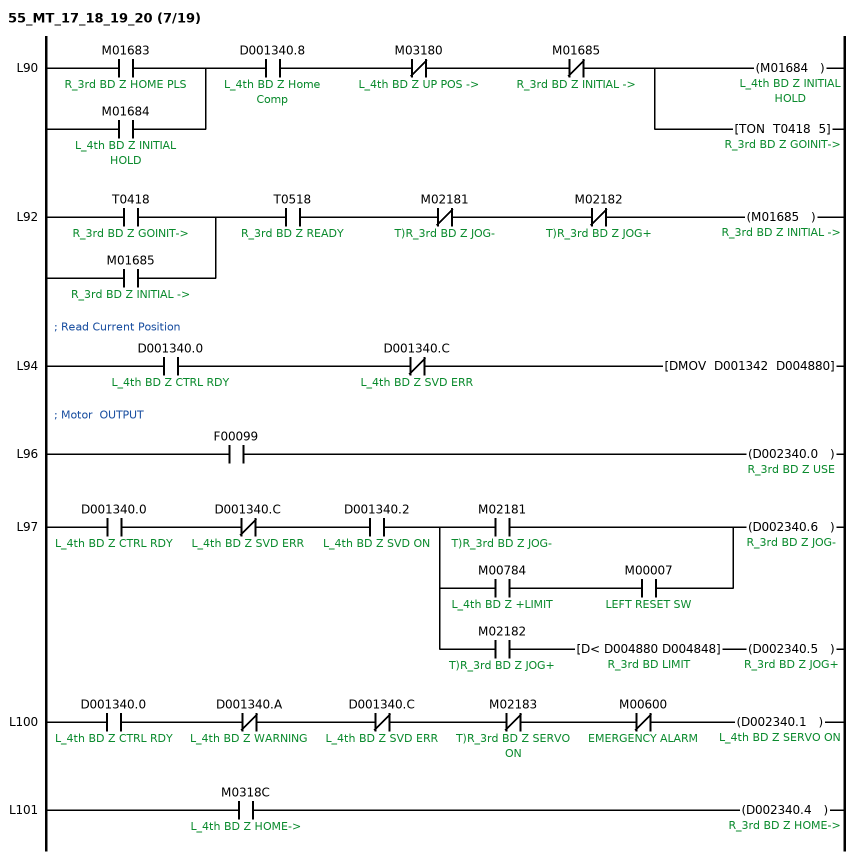
[picture p312: 55_MT_17_18_19_20 rungs L90-L101]
; L90
LOAD      M01683	// R_3rd BD Z HOME PLS
OR        M01684	// L_4th BD Z INITIAL HOLD
AND       D001340.8	// L_4th BD Z Home Comp
AND NOT   M03180	// L_4th BD Z UP POS ->
AND NOT   M01685	// R_3rd BD Z INITIAL ->
OUT       M01684	// L_4th BD Z INITIAL HOLD
TON       T0418 5	// R_3rd BD Z GOINIT->
; L92
LOAD      T0418	// R_3rd BD Z GOINIT->
OR        M01685	// R_3rd BD Z INITIAL ->
AND       T0518	// R_3rd BD Z READY
AND NOT   M02181	// T)R_3rd BD Z JOG-
AND NOT   M02182	// T)R_3rd BD Z JOG+
OUT       M01685	// R_3rd BD Z INITIAL ->
; L94
LOAD      D001340.0	// L_4th BD Z CTRL RDY
AND NOT   D001340.C	// L_4th BD Z SVD ERR
DMOV      D001342 D004880
// output comment: Read Current Position
//  Motor  OUTPUT
; L96
LOAD      F00099
OUT       D002340.0	// R_3rd BD Z USE
; L97
LOAD      D001340.0	// L_4th BD Z CTRL RDY
AND NOT   D001340.C	// L_4th BD Z SVD ERR
AND       D001340.2	// L_4th BD Z SVD ON
MPUSH
LOAD      M02181	// T)R_3rd BD Z JOG-
LOAD      M00784	// L_4th BD Z +LIMIT
AND       M00007	// LEFT RESET SW
OR LOAD
AND LOAD
OUT       D002340.6	// R_3rd BD Z JOG-
MPOP
AND       M02182	// T)R_3rd BD Z JOG+
ANDD<     D004880 D004848	// R_3rd BD LIMIT
OUT       D002340.5	// R_3rd BD Z JOG+
; L100
LOAD      D001340.0	// L_4th BD Z CTRL RDY
AND NOT   D001340.A	// L_4th BD Z WARNING
AND NOT   D001340.C	// L_4th BD Z SVD ERR
AND NOT   M02183	// T)R_3rd BD Z SERVO ON
AND NOT   M00600	// EMERGENCY ALARM
OUT       D002340.1	// L_4th BD Z SERVO ON
; L101
LOAD      M0318C	// L_4th BD Z HOME->
OUT       D002340.4	// R_3rd BD Z HOME->

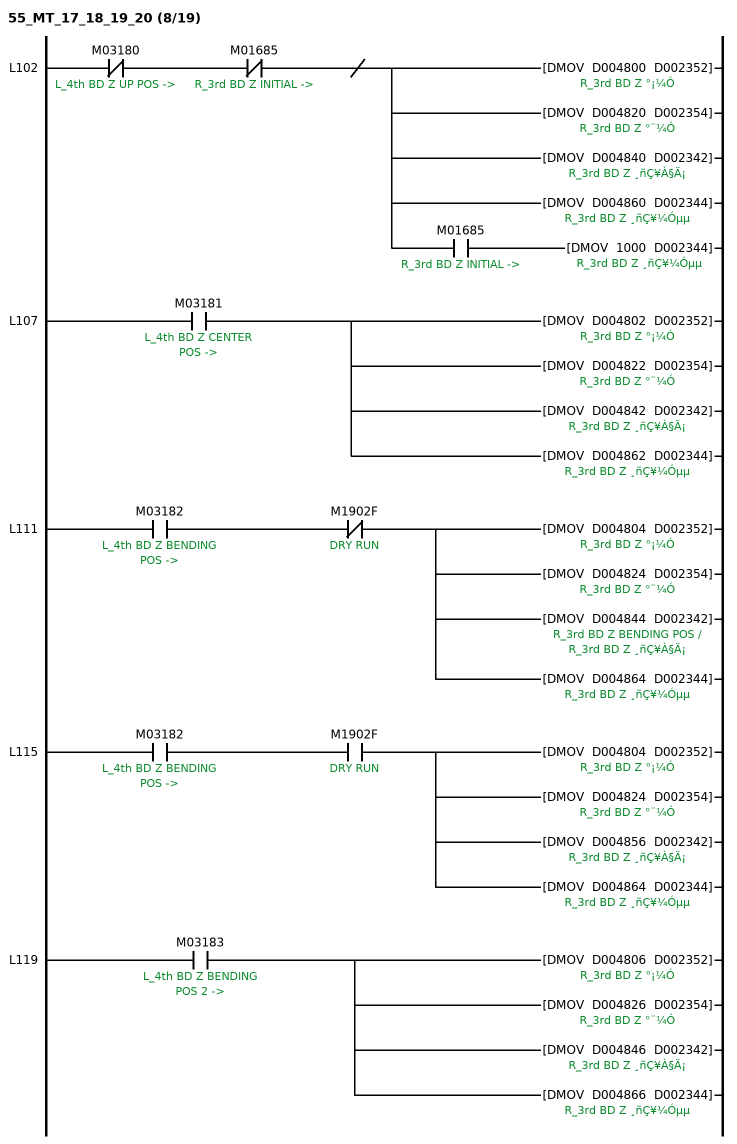
; L102
LOAD NOT  M03180	// L_4th BD Z UP POS ->
AND NOT   M01685	// R_3rd BD Z INITIAL ->
NOT
DMOV      D004800 D002352	// R_3rd BD Z °¡¼Ó
DMOV      D004820 D002354	// R_3rd BD Z °¨¼Ó
DMOV      D004840 D002342	// R_3rd BD Z ¸ñÇ¥À§Ä¡
DMOV      D004860 D002344	// R_3rd BD Z ¸ñÇ¥¼Óµµ
AND       M01685	// R_3rd BD Z INITIAL ->
DMOV      1000 D002344	// R_3rd BD Z ¸ñÇ¥¼Óµµ
; L107
LOAD      M03181	// L_4th BD Z CENTER POS ->
DMOV      D004802 D002352	// R_3rd BD Z °¡¼Ó
DMOV      D004822 D002354	// R_3rd BD Z °¨¼Ó
DMOV      D004842 D002342	// R_3rd BD Z ¸ñÇ¥À§Ä¡
DMOV      D004862 D002344	// R_3rd BD Z ¸ñÇ¥¼Óµµ
; L111
LOAD      M03182	// L_4th BD Z BENDING POS ->
AND NOT   M1902F	// DRY RUN
DMOV      D004804 D002352	// R_3rd BD Z °¡¼Ó
DMOV      D004824 D002354	// R_3rd BD Z °¨¼Ó
DMOV      D004844 D002342	// R_3rd BD Z BENDING POS / R_3rd BD Z ¸ñÇ¥À§Ä¡
DMOV      D004864 D002344	// R_3rd BD Z ¸ñÇ¥¼Óµµ
; L115
LOAD      M03182	// L_4th BD Z BENDING POS ->
AND       M1902F	// DRY RUN
DMOV      D004804 D002352	// R_3rd BD Z °¡¼Ó
DMOV      D004824 D002354	// R_3rd BD Z °¨¼Ó
DMOV      D004856 D002342	// R_3rd BD Z ¸ñÇ¥À§Ä¡
DMOV      D004864 D002344	// R_3rd BD Z ¸ñÇ¥¼Óµµ
; L119
LOAD      M03183	// L_4th BD Z BENDING POS 2 ->
DMOV      D004806 D002352	// R_3rd BD Z °¡¼Ó
DMOV      D004826 D002354	// R_3rd BD Z °¨¼Ó
DMOV      D004846 D002342	// R_3rd BD Z ¸ñÇ¥À§Ä¡
DMOV      D004866 D002344	// R_3rd BD Z ¸ñÇ¥¼Óµµ

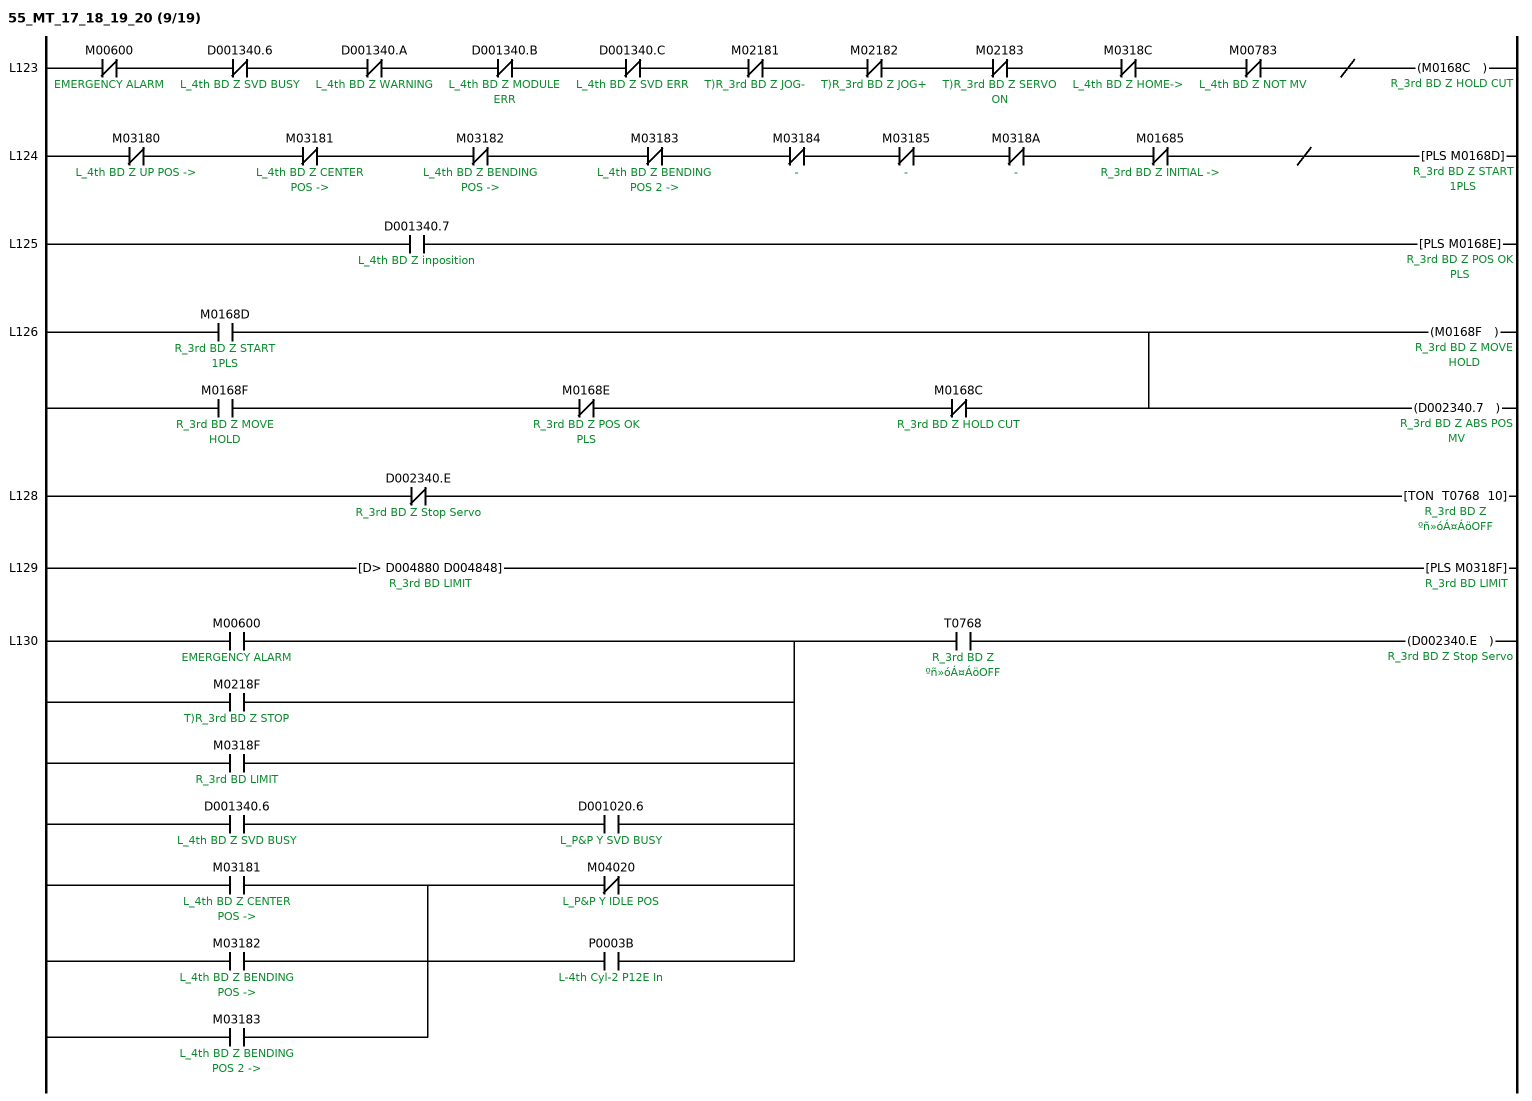
; L123
LOAD NOT  M00600	// EMERGENCY ALARM
AND NOT   D001340.6	// L_4th BD Z SVD BUSY
AND NOT   D001340.A	// L_4th BD Z WARNING
AND NOT   D001340.B	// L_4th BD Z MODULE ERR
AND NOT   D001340.C	// L_4th BD Z SVD ERR
AND NOT   M02181	// T)R_3rd BD Z JOG-
AND NOT   M02182	// T)R_3rd BD Z JOG+
AND NOT   M02183	// T)R_3rd BD Z SERVO ON
AND NOT   M0318C	// L_4th BD Z HOME->
AND NOT   M00783	// L_4th BD Z NOT MV
NOT
OUT       M0168C	// R_3rd BD Z HOLD CUT
; L124
LOAD NOT  M03180	// L_4th BD Z UP POS ->
AND NOT   M03181	// L_4th BD Z CENTER POS ->
AND NOT   M03182	// L_4th BD Z BENDING POS ->
AND NOT   M03183	// L_4th BD Z BENDING POS 2 ->
AND NOT   M03184	// -
AND NOT   M03185	// -
AND NOT   M0318A	// -
AND NOT   M01685	// R_3rd BD Z INITIAL ->
NOT
OUTP      M0168D	// R_3rd BD Z START 1PLS
; L125
LOAD      D001340.7	// L_4th BD Z inposition
OUTP      M0168E	// R_3rd BD Z POS OK PLS
; L126
LOAD      M0168D	// R_3rd BD Z START 1PLS
LOAD      M0168F	// R_3rd BD Z MOVE HOLD
AND NOT   M0168E	// R_3rd BD Z POS OK PLS
AND NOT   M0168C	// R_3rd BD Z HOLD CUT
OR LOAD
OUT       M0168F	// R_3rd BD Z MOVE HOLD
OUT       D002340.7	// R_3rd BD Z ABS POS MV
; L128
LOAD NOT  D002340.E	// R_3rd BD Z Stop Servo
TON       T0768 10	// R_3rd BD Z ºñ»óÁ¤ÁöOFF
; L129
LOADD>    D004880 D004848	// R_3rd BD LIMIT
OUTP      M0318F	// R_3rd BD LIMIT
; L130
LOAD      M00600	// EMERGENCY ALARM
OR        M0218F	// T)R_3rd BD Z STOP
OR        M0318F	// R_3rd BD LIMIT
LOAD      D001340.6	// L_4th BD Z SVD BUSY
AND       D001020.6	// L_P&P Y SVD BUSY
OR LOAD
LOAD      M03181	// L_4th BD Z CENTER POS ->
OR        M03182	// L_4th BD Z BENDING POS ->
OR        M03183	// L_4th BD Z BENDING POS 2 ->
LOAD NOT  M04020	// L_P&P Y IDLE POS
OR        P0003B	// L-4th Cyl-2 P12E In
AND LOAD
OR LOAD
AND       T0768	// R_3rd BD Z ºñ»óÁ¤ÁöOFF
OUT       D002340.E	// R_3rd BD Z Stop Servo

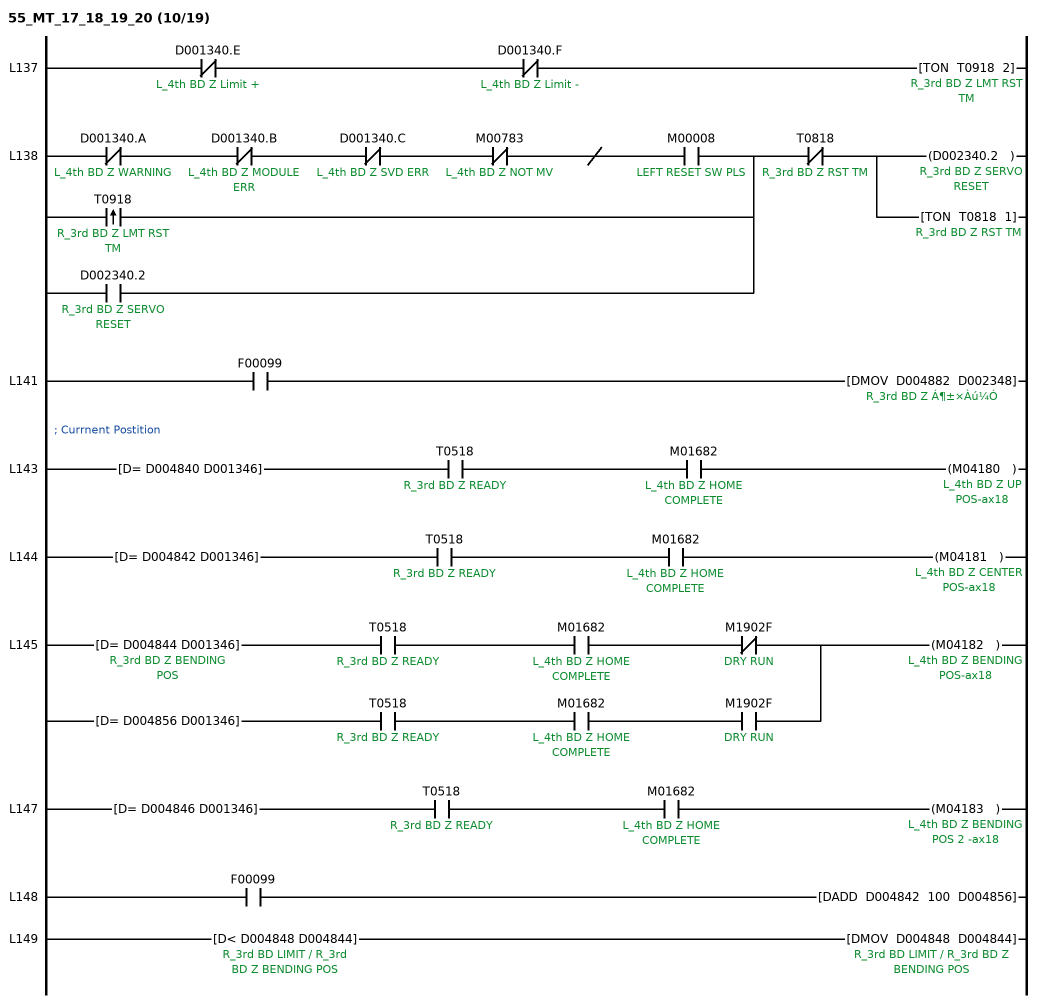
; L137
LOAD NOT  D001340.E	// L_4th BD Z Limit +
AND NOT   D001340.F	// L_4th BD Z Limit -
TON       T0918 2	// R_3rd BD Z LMT RST TM
; L138
LOAD NOT  D001340.A	// L_4th BD Z WARNING
AND NOT   D001340.B	// L_4th BD Z MODULE ERR
AND NOT   D001340.C	// L_4th BD Z SVD ERR
AND NOT   M00783	// L_4th BD Z NOT MV
NOT
AND       M00008	// LEFT RESET SW PLS
ORP       T0918	// R_3rd BD Z LMT RST TM
OR        D002340.2	// R_3rd BD Z SERVO RESET
AND NOT   T0818	// R_3rd BD Z RST TM
OUT       D002340.2	// R_3rd BD Z SERVO RESET
TON       T0818 1	// R_3rd BD Z RST TM
; L141
LOAD      F00099
DMOV      D004882 D002348	// R_3rd BD Z Á¶±×Àú¼Ó
// Currnent Postition
; L143
LOADD=    D004840 D001346
AND       T0518	// R_3rd BD Z READY
AND       M01682	// L_4th BD Z HOME COMPLETE
OUT       M04180	// L_4th BD Z UP POS-ax18
; L144
LOADD=    D004842 D001346
AND       T0518	// R_3rd BD Z READY
AND       M01682	// L_4th BD Z HOME COMPLETE
OUT       M04181	// L_4th BD Z CENTER POS-ax18
; L145
LOADD=    D004844 D001346	// R_3rd BD Z BENDING POS
AND       T0518	// R_3rd BD Z READY
AND       M01682	// L_4th BD Z HOME COMPLETE
AND NOT   M1902F	// DRY RUN
LOADD=    D004856 D001346
AND       T0518	// R_3rd BD Z READY
AND       M01682	// L_4th BD Z HOME COMPLETE
AND       M1902F	// DRY RUN
OR LOAD
OUT       M04182	// L_4th BD Z BENDING POS-ax18
; L147
LOADD=    D004846 D001346
AND       T0518	// R_3rd BD Z READY
AND       M01682	// L_4th BD Z HOME COMPLETE
OUT       M04183	// L_4th BD Z BENDING POS 2 -ax18
; L148
LOAD      F00099
DADD      D004842 100 D004856
; L149
LOADD<    D004848 D004844	// R_3rd BD LIMIT / R_3rd BD Z BENDING POS
DMOV      D004848 D004844	// R_3rd BD LIMIT / R_3rd BD Z BENDING POS

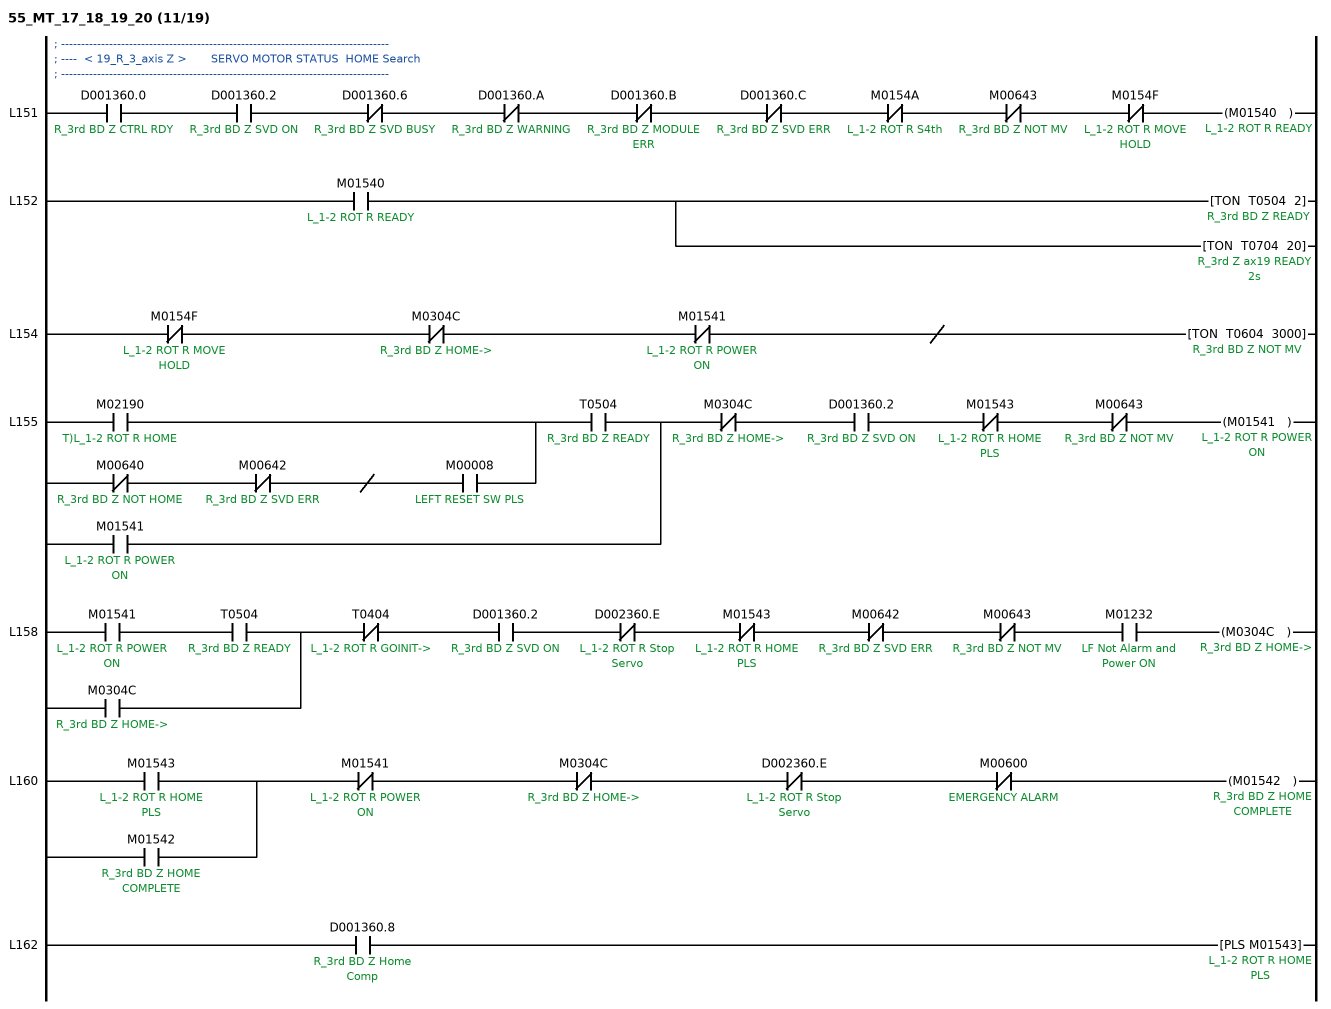
// ----------------------------------------------------------------------------------
// 
// ----  < 19_R_3_axis Z >       SERVO MOTOR STATUS  HOME Search
// 
// ----------------------------------------------------------------------------------
; L151
LOAD      D001360.0	// R_3rd BD Z CTRL RDY
AND       D001360.2	// R_3rd BD Z SVD ON
AND NOT   D001360.6	// R_3rd BD Z SVD BUSY
AND NOT   D001360.A	// R_3rd BD Z WARNING
AND NOT   D001360.B	// R_3rd BD Z MODULE ERR
AND NOT   D001360.C	// R_3rd BD Z SVD ERR
AND NOT   M0154A	// L_1-2 ROT R S4th
AND NOT   M00643	// R_3rd BD Z NOT MV
AND NOT   M0154F	// L_1-2 ROT R MOVE HOLD
OUT       M01540	// L_1-2 ROT R READY
; L152
LOAD      M01540	// L_1-2 ROT R READY
TON       T0504 2	// R_3rd BD Z READY
TON       T0704 20	// R_3rd Z ax19 READY 2s
; L154
LOAD NOT  M0154F	// L_1-2 ROT R MOVE HOLD
AND NOT   M0304C	// R_3rd BD Z HOME->
AND NOT   M01541	// L_1-2 ROT R POWER ON
NOT
TON       T0604 3000	// R_3rd BD Z NOT MV
; L155
LOAD      M02190	// T)L_1-2 ROT R HOME
LOAD NOT  M00640	// R_3rd BD Z NOT HOME
AND NOT   M00642	// R_3rd BD Z SVD ERR
NOT
AND       M00008	// LEFT RESET SW PLS
OR LOAD
AND       T0504	// R_3rd BD Z READY
OR        M01541	// L_1-2 ROT R POWER ON
AND NOT   M0304C	// R_3rd BD Z HOME->
AND       D001360.2	// R_3rd BD Z SVD ON
AND NOT   M01543	// L_1-2 ROT R HOME PLS
AND NOT   M00643	// R_3rd BD Z NOT MV
OUT       M01541	// L_1-2 ROT R POWER ON
; L158
LOAD      M01541	// L_1-2 ROT R POWER ON
AND       T0504	// R_3rd BD Z READY
OR        M0304C	// R_3rd BD Z HOME->
AND NOT   T0404	// L_1-2 ROT R GOINIT->
AND       D001360.2	// R_3rd BD Z SVD ON
AND NOT   D002360.E	// L_1-2 ROT R Stop Servo
AND NOT   M01543	// L_1-2 ROT R HOME PLS
AND NOT   M00642	// R_3rd BD Z SVD ERR
AND NOT   M00643	// R_3rd BD Z NOT MV
AND       M01232	// LF Not Alarm and Power ON
OUT       M0304C	// R_3rd BD Z HOME->
; L160
LOAD      M01543	// L_1-2 ROT R HOME PLS
OR        M01542	// R_3rd BD Z HOME COMPLETE
AND NOT   M01541	// L_1-2 ROT R POWER ON
AND NOT   M0304C	// R_3rd BD Z HOME->
AND NOT   D002360.E	// L_1-2 ROT R Stop Servo
AND NOT   M00600	// EMERGENCY ALARM
OUT       M01542	// R_3rd BD Z HOME COMPLETE
; L162
LOAD      D001360.8	// R_3rd BD Z Home Comp
OUTP      M01543	// L_1-2 ROT R HOME PLS

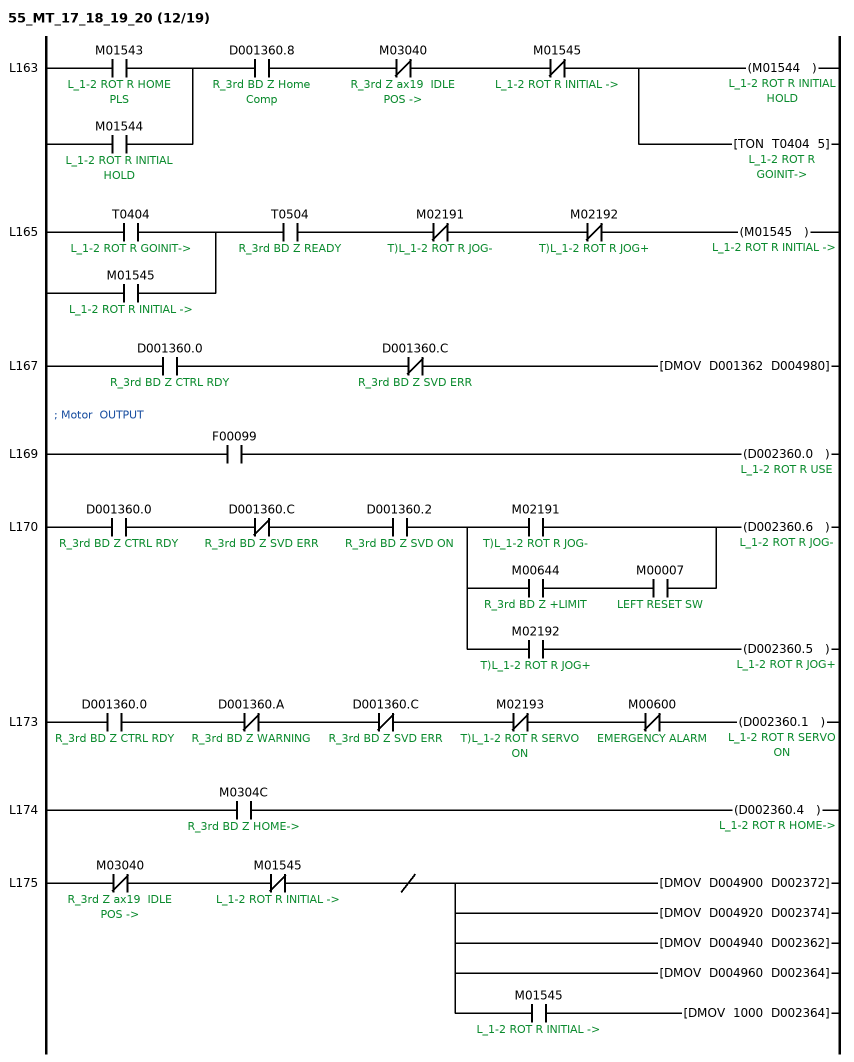
; L163
LOAD      M01543	// L_1-2 ROT R HOME PLS
OR        M01544	// L_1-2 ROT R INITIAL HOLD
AND       D001360.8	// R_3rd BD Z Home Comp
AND NOT   M03040	// R_3rd Z ax19  IDLE POS ->
AND NOT   M01545	// L_1-2 ROT R INITIAL ->
OUT       M01544	// L_1-2 ROT R INITIAL HOLD
TON       T0404 5	// L_1-2 ROT R GOINIT->
; L165
LOAD      T0404	// L_1-2 ROT R GOINIT->
OR        M01545	// L_1-2 ROT R INITIAL ->
AND       T0504	// R_3rd BD Z READY
AND NOT   M02191	// T)L_1-2 ROT R JOG-
AND NOT   M02192	// T)L_1-2 ROT R JOG+
OUT       M01545	// L_1-2 ROT R INITIAL ->
; L167
LOAD      D001360.0	// R_3rd BD Z CTRL RDY
AND NOT   D001360.C	// R_3rd BD Z SVD ERR
DMOV      D001362 D004980
//  Motor  OUTPUT
; L169
LOAD      F00099
OUT       D002360.0	// L_1-2 ROT R USE
; L170
LOAD      D001360.0	// R_3rd BD Z CTRL RDY
AND NOT   D001360.C	// R_3rd BD Z SVD ERR
AND       D001360.2	// R_3rd BD Z SVD ON
MPUSH
LOAD      M02191	// T)L_1-2 ROT R JOG-
LOAD      M00644	// R_3rd BD Z +LIMIT
AND       M00007	// LEFT RESET SW
OR LOAD
AND LOAD
OUT       D002360.6	// L_1-2 ROT R JOG-
MPOP
AND       M02192	// T)L_1-2 ROT R JOG+
OUT       D002360.5	// L_1-2 ROT R JOG+
; L173
LOAD      D001360.0	// R_3rd BD Z CTRL RDY
AND NOT   D001360.A	// R_3rd BD Z WARNING
AND NOT   D001360.C	// R_3rd BD Z SVD ERR
AND NOT   M02193	// T)L_1-2 ROT R SERVO ON
AND NOT   M00600	// EMERGENCY ALARM
OUT       D002360.1	// L_1-2 ROT R SERVO ON
; L174
LOAD      M0304C	// R_3rd BD Z HOME->
OUT       D002360.4	// L_1-2 ROT R HOME->
; L175
LOAD NOT  M03040	// R_3rd Z ax19  IDLE POS ->
AND NOT   M01545	// L_1-2 ROT R INITIAL ->
NOT
DMOV      D004900 D002372
DMOV      D004920 D002374
DMOV      D004940 D002362
DMOV      D004960 D002364
AND       M01545	// L_1-2 ROT R INITIAL ->
DMOV      1000 D002364

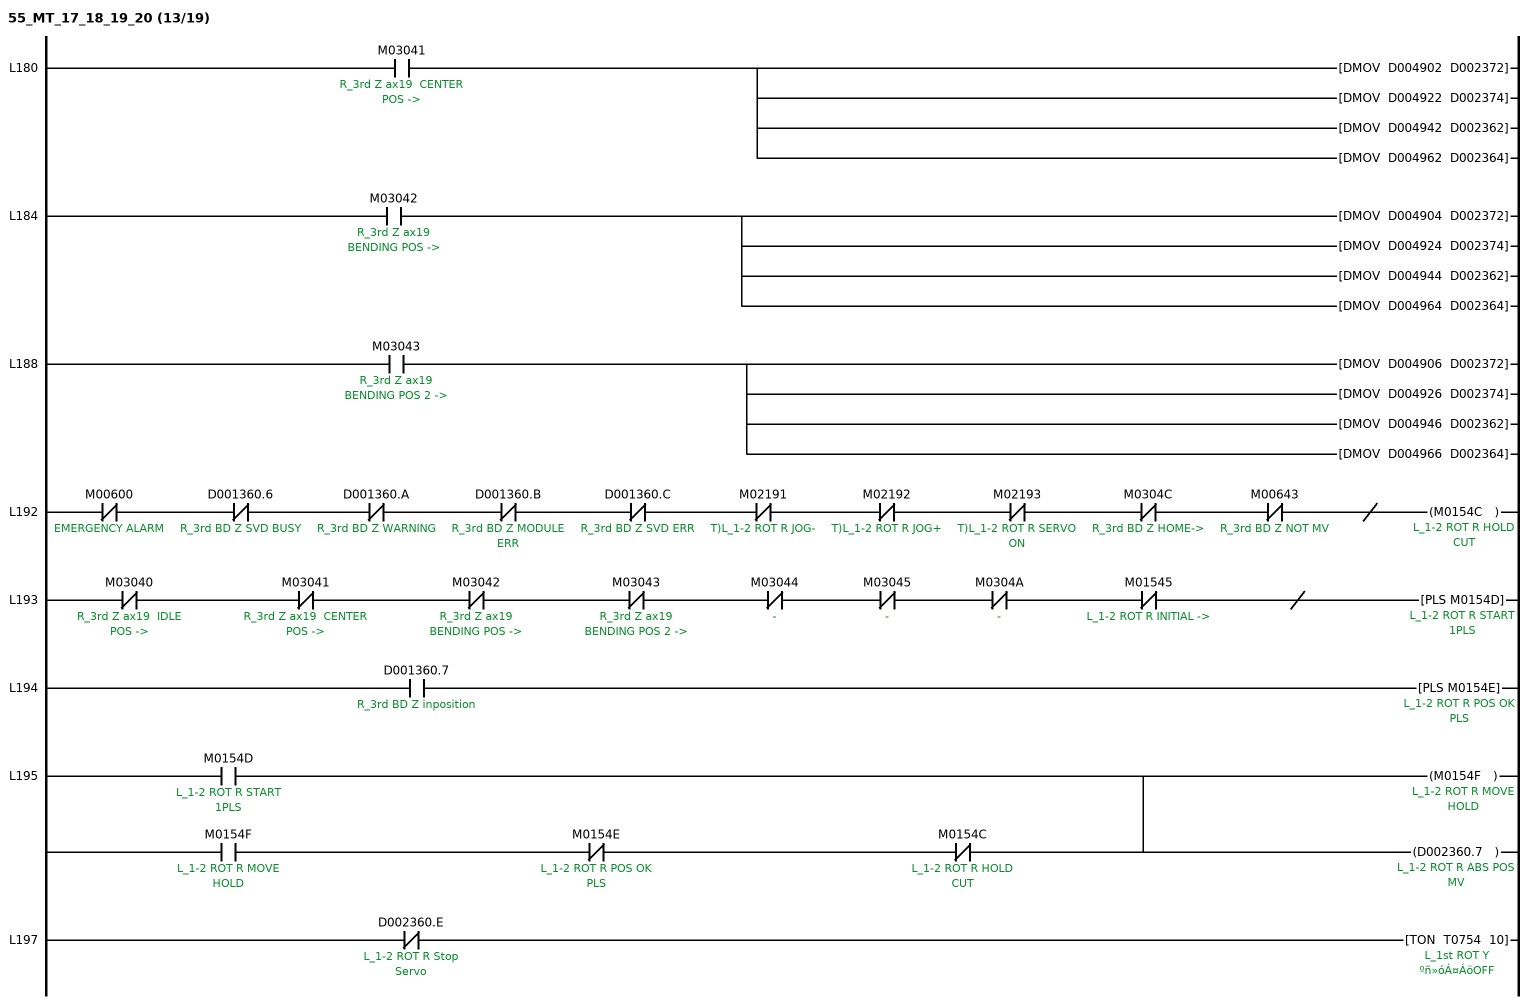
; L180
LOAD      M03041	// R_3rd Z ax19  CENTER POS ->
DMOV      D004902 D002372
DMOV      D004922 D002374
DMOV      D004942 D002362
DMOV      D004962 D002364
; L184
LOAD      M03042	// R_3rd Z ax19  BENDING POS ->
DMOV      D004904 D002372
DMOV      D004924 D002374
DMOV      D004944 D002362
DMOV      D004964 D002364
; L188
LOAD      M03043	// R_3rd Z ax19 BENDING POS 2 ->
DMOV      D004906 D002372
DMOV      D004926 D002374
DMOV      D004946 D002362
DMOV      D004966 D002364
; L192
LOAD NOT  M00600	// EMERGENCY ALARM
AND NOT   D001360.6	// R_3rd BD Z SVD BUSY
AND NOT   D001360.A	// R_3rd BD Z WARNING
AND NOT   D001360.B	// R_3rd BD Z MODULE ERR
AND NOT   D001360.C	// R_3rd BD Z SVD ERR
AND NOT   M02191	// T)L_1-2 ROT R JOG-
AND NOT   M02192	// T)L_1-2 ROT R JOG+
AND NOT   M02193	// T)L_1-2 ROT R SERVO ON
AND NOT   M0304C	// R_3rd BD Z HOME->
AND NOT   M00643	// R_3rd BD Z NOT MV
NOT
OUT       M0154C	// L_1-2 ROT R HOLD CUT
; L193
LOAD NOT  M03040	// R_3rd Z ax19  IDLE POS ->
AND NOT   M03041	// R_3rd Z ax19  CENTER POS ->
AND NOT   M03042	// R_3rd Z ax19  BENDING POS ->
AND NOT   M03043	// R_3rd Z ax19 BENDING POS 2 ->
AND NOT   M03044	// -
AND NOT   M03045	// -
AND NOT   M0304A	// -
AND NOT   M01545	// L_1-2 ROT R INITIAL ->
NOT
OUTP      M0154D	// L_1-2 ROT R START 1PLS
; L194
LOAD      D001360.7	// R_3rd BD Z inposition
OUTP      M0154E	// L_1-2 ROT R POS OK PLS
; L195
LOAD      M0154D	// L_1-2 ROT R START 1PLS
LOAD      M0154F	// L_1-2 ROT R MOVE HOLD
AND NOT   M0154E	// L_1-2 ROT R POS OK PLS
AND NOT   M0154C	// L_1-2 ROT R HOLD CUT
OR LOAD
OUT       M0154F	// L_1-2 ROT R MOVE HOLD
OUT       D002360.7	// L_1-2 ROT R ABS POS MV
; L197
LOAD NOT  D002360.E	// L_1-2 ROT R Stop Servo
TON       T0754 10	// L_1st ROT Y ºñ»óÁ¤ÁöOFF

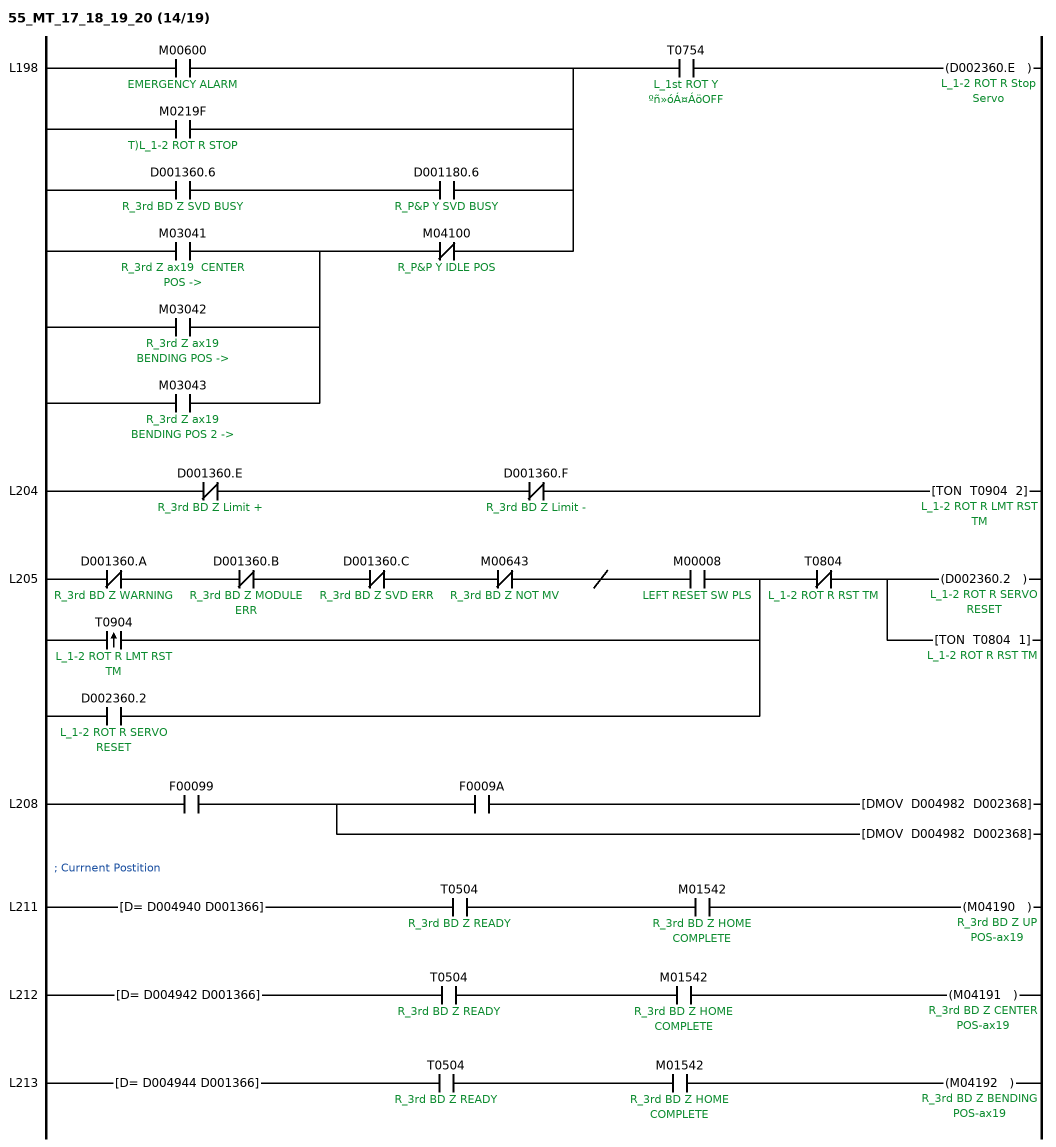
; L198
LOAD      M00600	// EMERGENCY ALARM
OR        M0219F	// T)L_1-2 ROT R STOP
LOAD      D001360.6	// R_3rd BD Z SVD BUSY
AND       D001180.6	// R_P&P Y SVD BUSY
OR LOAD
LOAD      M03041	// R_3rd Z ax19  CENTER POS ->
OR        M03042	// R_3rd Z ax19  BENDING POS ->
OR        M03043	// R_3rd Z ax19 BENDING POS 2 ->
AND NOT   M04100	// R_P&P Y IDLE POS
OR LOAD
AND       T0754	// L_1st ROT Y ºñ»óÁ¤ÁöOFF
OUT       D002360.E	// L_1-2 ROT R Stop Servo
; L204
LOAD NOT  D001360.E	// R_3rd BD Z Limit +
AND NOT   D001360.F	// R_3rd BD Z Limit -
TON       T0904 2	// L_1-2 ROT R LMT RST TM
; L205
LOAD NOT  D001360.A	// R_3rd BD Z WARNING
AND NOT   D001360.B	// R_3rd BD Z MODULE ERR
AND NOT   D001360.C	// R_3rd BD Z SVD ERR
AND NOT   M00643	// R_3rd BD Z NOT MV
NOT
AND       M00008	// LEFT RESET SW PLS
ORP       T0904	// L_1-2 ROT R LMT RST TM
OR        D002360.2	// L_1-2 ROT R SERVO RESET
AND NOT   T0804	// L_1-2 ROT R RST TM
OUT       D002360.2	// L_1-2 ROT R SERVO RESET
TON       T0804 1	// L_1-2 ROT R RST TM
; L208
LOAD      F00099
MPUSH
AND       F0009A
DMOV      D004982 D002368
MPOP
DMOV      D004982 D002368
// Currnent Postition
; L211
LOADD=    D004940 D001366
AND       T0504	// R_3rd BD Z READY
AND       M01542	// R_3rd BD Z HOME COMPLETE
OUT       M04190	// R_3rd BD Z UP POS-ax19
; L212
LOADD=    D004942 D001366
AND       T0504	// R_3rd BD Z READY
AND       M01542	// R_3rd BD Z HOME COMPLETE
OUT       M04191	// R_3rd BD Z CENTER POS-ax19
; L213
LOADD=    D004944 D001366
AND       T0504	// R_3rd BD Z READY
AND       M01542	// R_3rd BD Z HOME COMPLETE
OUT       M04192	// R_3rd BD Z BENDING POS-ax19

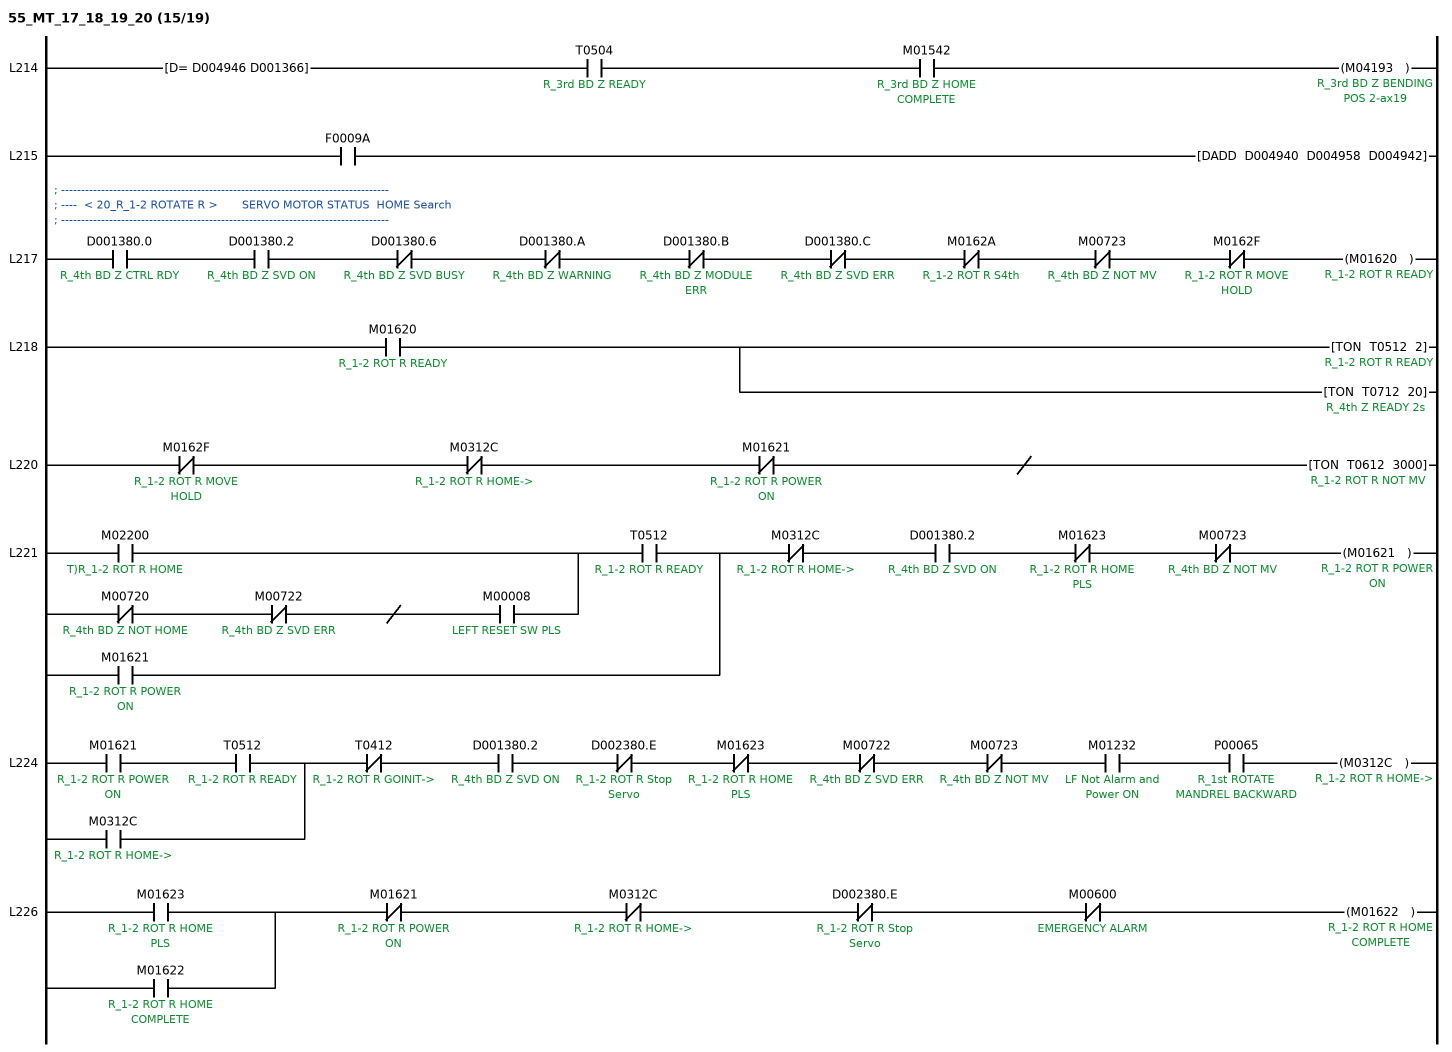
; L214
LOADD=    D004946 D001366
AND       T0504	// R_3rd BD Z READY
AND       M01542	// R_3rd BD Z HOME COMPLETE
OUT       M04193	// R_3rd BD Z BENDING POS 2-ax19
; L215
LOAD      F0009A
DADD      D004940 D004958 D004942
// ----------------------------------------------------------------------------------
// 
// ----  < 20_R_1-2 ROTATE R >       SERVO MOTOR STATUS  HOME Search
// 
// ----------------------------------------------------------------------------------
; L217
LOAD      D001380.0	// R_4th BD Z CTRL RDY
AND       D001380.2	// R_4th BD Z SVD ON
AND NOT   D001380.6	// R_4th BD Z SVD BUSY
AND NOT   D001380.A	// R_4th BD Z WARNING
AND NOT   D001380.B	// R_4th BD Z MODULE ERR
AND NOT   D001380.C	// R_4th BD Z SVD ERR
AND NOT   M0162A	// R_1-2 ROT R S4th
AND NOT   M00723	// R_4th BD Z NOT MV
AND NOT   M0162F	// R_1-2 ROT R MOVE HOLD
OUT       M01620	// R_1-2 ROT R READY
; L218
LOAD      M01620	// R_1-2 ROT R READY
TON       T0512 2	// R_1-2 ROT R READY
TON       T0712 20	// R_4th Z READY 2s
; L220
LOAD NOT  M0162F	// R_1-2 ROT R MOVE HOLD
AND NOT   M0312C	// R_1-2 ROT R HOME->
AND NOT   M01621	// R_1-2 ROT R POWER ON
NOT
TON       T0612 3000	// R_1-2 ROT R NOT MV
; L221
LOAD      M02200	// T)R_1-2 ROT R HOME
LOAD NOT  M00720	// R_4th BD Z NOT HOME
AND NOT   M00722	// R_4th BD Z SVD ERR
NOT
AND       M00008	// LEFT RESET SW PLS
OR LOAD
AND       T0512	// R_1-2 ROT R READY
OR        M01621	// R_1-2 ROT R POWER ON
AND NOT   M0312C	// R_1-2 ROT R HOME->
AND       D001380.2	// R_4th BD Z SVD ON
AND NOT   M01623	// R_1-2 ROT R HOME PLS
AND NOT   M00723	// R_4th BD Z NOT MV
OUT       M01621	// R_1-2 ROT R POWER ON
; L224
LOAD      M01621	// R_1-2 ROT R POWER ON
AND       T0512	// R_1-2 ROT R READY
OR        M0312C	// R_1-2 ROT R HOME->
AND NOT   T0412	// R_1-2 ROT R GOINIT->
AND       D001380.2	// R_4th BD Z SVD ON
AND NOT   D002380.E	// R_1-2 ROT R Stop Servo
AND NOT   M01623	// R_1-2 ROT R HOME PLS
AND NOT   M00722	// R_4th BD Z SVD ERR
AND NOT   M00723	// R_4th BD Z NOT MV
AND       M01232	// LF Not Alarm and Power ON
AND       P00065	// R_1st ROTATE MANDREL BACKWARD
OUT       M0312C	// R_1-2 ROT R HOME->
; L226
LOAD      M01623	// R_1-2 ROT R HOME PLS
OR        M01622	// R_1-2 ROT R HOME COMPLETE
AND NOT   M01621	// R_1-2 ROT R POWER ON
AND NOT   M0312C	// R_1-2 ROT R HOME->
AND NOT   D002380.E	// R_1-2 ROT R Stop Servo
AND NOT   M00600	// EMERGENCY ALARM
OUT       M01622	// R_1-2 ROT R HOME COMPLETE

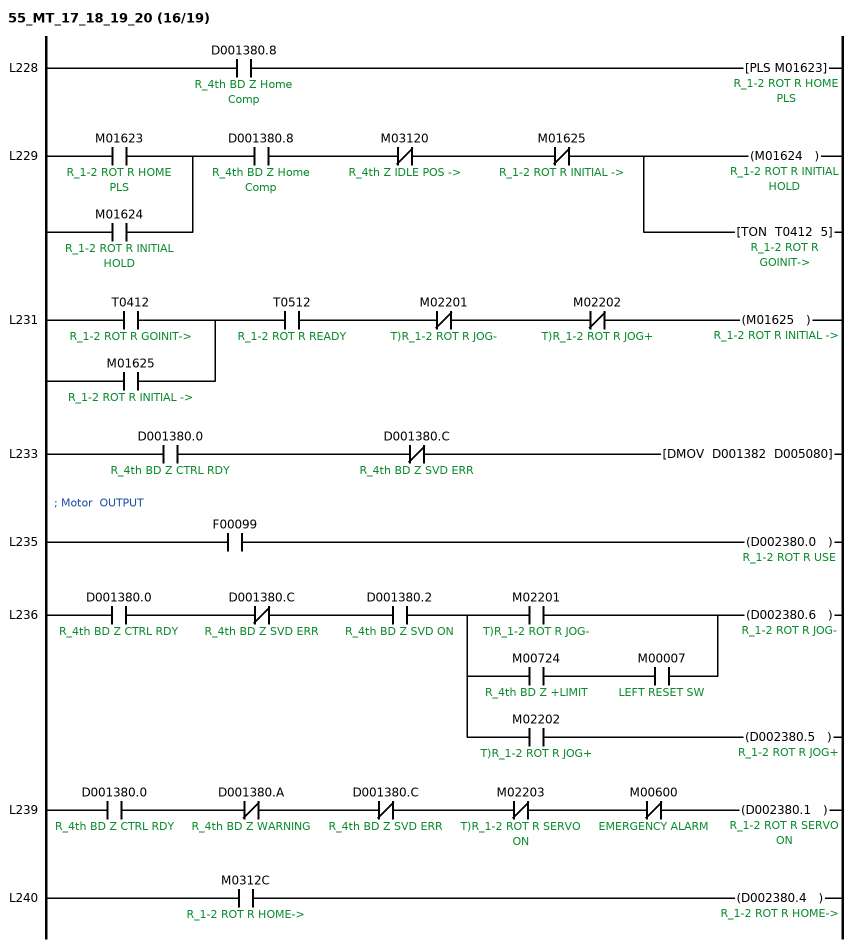
; L228
LOAD      D001380.8	// R_4th BD Z Home Comp
OUTP      M01623	// R_1-2 ROT R HOME PLS
; L229
LOAD      M01623	// R_1-2 ROT R HOME PLS
OR        M01624	// R_1-2 ROT R INITIAL HOLD
AND       D001380.8	// R_4th BD Z Home Comp
AND NOT   M03120	// R_4th Z IDLE POS ->
AND NOT   M01625	// R_1-2 ROT R INITIAL ->
OUT       M01624	// R_1-2 ROT R INITIAL HOLD
TON       T0412 5	// R_1-2 ROT R GOINIT->
; L231
LOAD      T0412	// R_1-2 ROT R GOINIT->
OR        M01625	// R_1-2 ROT R INITIAL ->
AND       T0512	// R_1-2 ROT R READY
AND NOT   M02201	// T)R_1-2 ROT R JOG-
AND NOT   M02202	// T)R_1-2 ROT R JOG+
OUT       M01625	// R_1-2 ROT R INITIAL ->
; L233
LOAD      D001380.0	// R_4th BD Z CTRL RDY
AND NOT   D001380.C	// R_4th BD Z SVD ERR
DMOV      D001382 D005080
//  Motor  OUTPUT
; L235
LOAD      F00099
OUT       D002380.0	// R_1-2 ROT R USE
; L236
LOAD      D001380.0	// R_4th BD Z CTRL RDY
AND NOT   D001380.C	// R_4th BD Z SVD ERR
AND       D001380.2	// R_4th BD Z SVD ON
MPUSH
LOAD      M02201	// T)R_1-2 ROT R JOG-
LOAD      M00724	// R_4th BD Z +LIMIT
AND       M00007	// LEFT RESET SW
OR LOAD
AND LOAD
OUT       D002380.6	// R_1-2 ROT R JOG-
MPOP
AND       M02202	// T)R_1-2 ROT R JOG+
OUT       D002380.5	// R_1-2 ROT R JOG+
; L239
LOAD      D001380.0	// R_4th BD Z CTRL RDY
AND NOT   D001380.A	// R_4th BD Z WARNING
AND NOT   D001380.C	// R_4th BD Z SVD ERR
AND NOT   M02203	// T)R_1-2 ROT R SERVO ON
AND NOT   M00600	// EMERGENCY ALARM
OUT       D002380.1	// R_1-2 ROT R SERVO ON
; L240
LOAD      M0312C	// R_1-2 ROT R HOME->
OUT       D002380.4	// R_1-2 ROT R HOME->

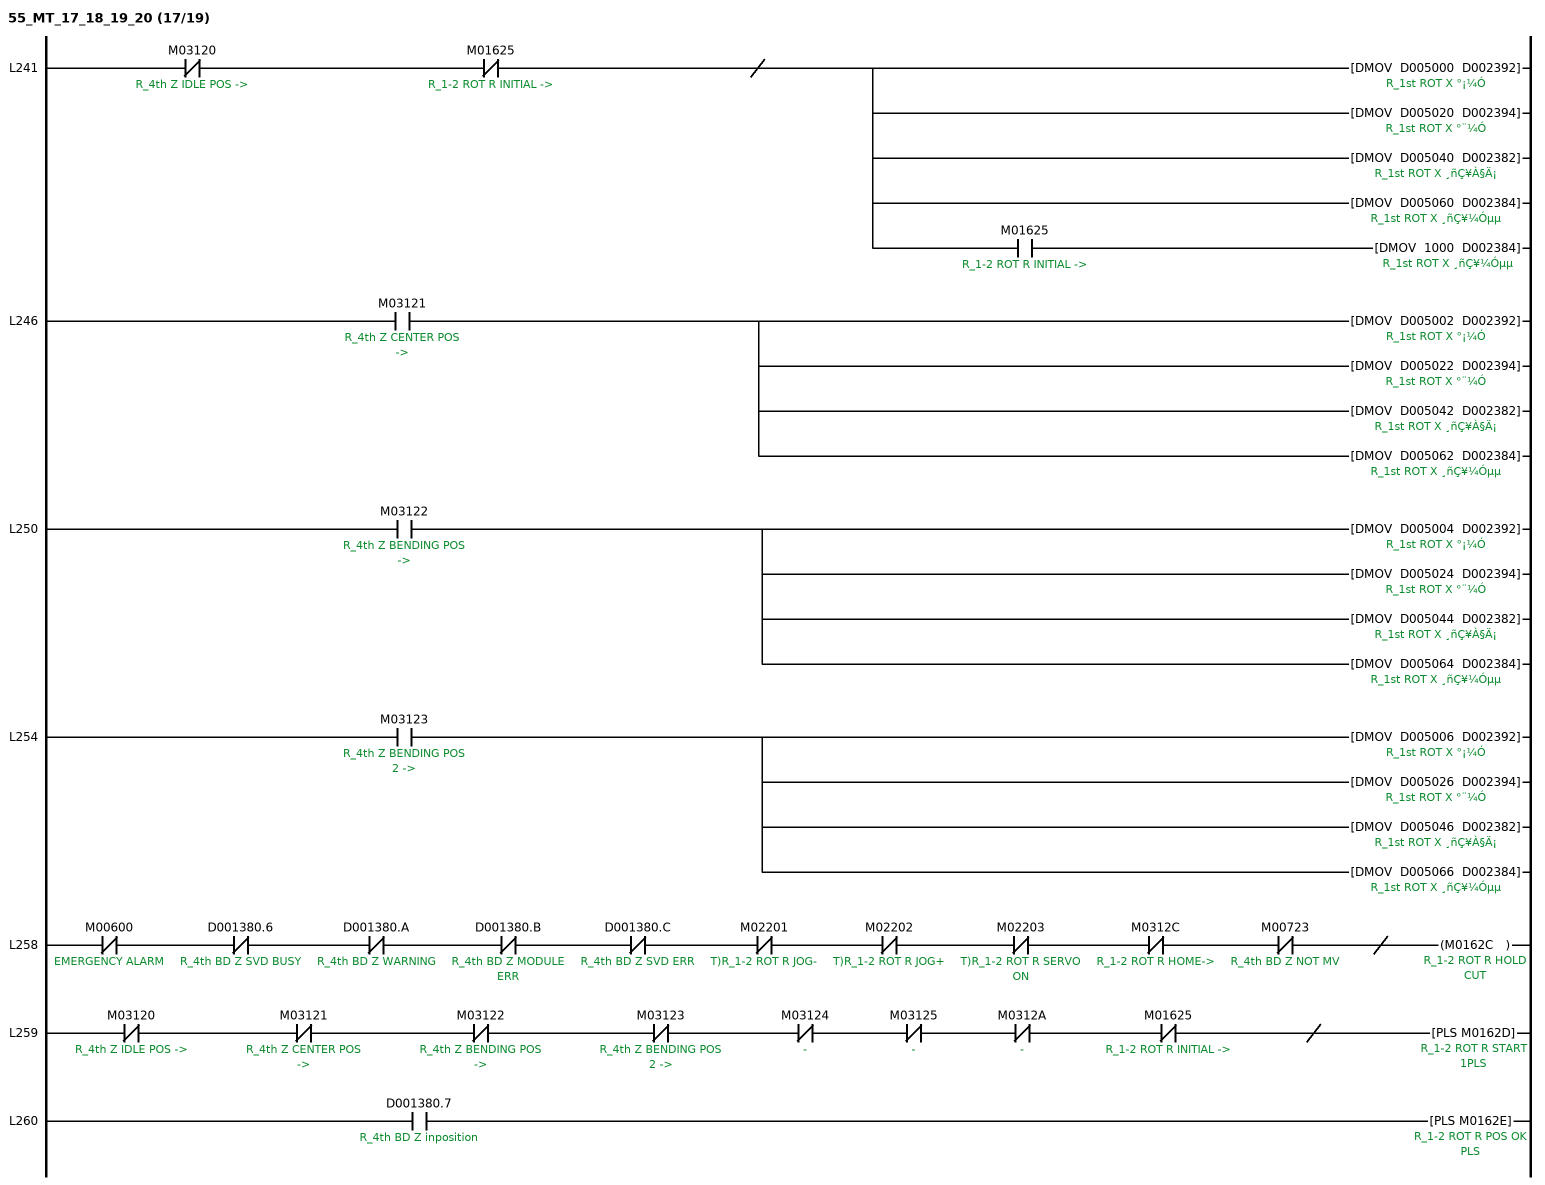
; L241
LOAD NOT  M03120	// R_4th Z IDLE POS ->
AND NOT   M01625	// R_1-2 ROT R INITIAL ->
NOT
DMOV      D005000 D002392	// R_1st ROT X °¡¼Ó
DMOV      D005020 D002394	// R_1st ROT X °¨¼Ó
DMOV      D005040 D002382	// R_1st ROT X ¸ñÇ¥À§Ä¡
DMOV      D005060 D002384	// R_1st ROT X ¸ñÇ¥¼Óµµ
AND       M01625	// R_1-2 ROT R INITIAL ->
DMOV      1000 D002384	// R_1st ROT X ¸ñÇ¥¼Óµµ
; L246
LOAD      M03121	// R_4th Z CENTER POS ->
DMOV      D005002 D002392	// R_1st ROT X °¡¼Ó
DMOV      D005022 D002394	// R_1st ROT X °¨¼Ó
DMOV      D005042 D002382	// R_1st ROT X ¸ñÇ¥À§Ä¡
DMOV      D005062 D002384	// R_1st ROT X ¸ñÇ¥¼Óµµ
; L250
LOAD      M03122	// R_4th Z BENDING POS ->
DMOV      D005004 D002392	// R_1st ROT X °¡¼Ó
DMOV      D005024 D002394	// R_1st ROT X °¨¼Ó
DMOV      D005044 D002382	// R_1st ROT X ¸ñÇ¥À§Ä¡
DMOV      D005064 D002384	// R_1st ROT X ¸ñÇ¥¼Óµµ
; L254
LOAD      M03123	// R_4th Z BENDING POS 2 ->
DMOV      D005006 D002392	// R_1st ROT X °¡¼Ó
DMOV      D005026 D002394	// R_1st ROT X °¨¼Ó
DMOV      D005046 D002382	// R_1st ROT X ¸ñÇ¥À§Ä¡
DMOV      D005066 D002384	// R_1st ROT X ¸ñÇ¥¼Óµµ
; L258
LOAD NOT  M00600	// EMERGENCY ALARM
AND NOT   D001380.6	// R_4th BD Z SVD BUSY
AND NOT   D001380.A	// R_4th BD Z WARNING
AND NOT   D001380.B	// R_4th BD Z MODULE ERR
AND NOT   D001380.C	// R_4th BD Z SVD ERR
AND NOT   M02201	// T)R_1-2 ROT R JOG-
AND NOT   M02202	// T)R_1-2 ROT R JOG+
AND NOT   M02203	// T)R_1-2 ROT R SERVO ON
AND NOT   M0312C	// R_1-2 ROT R HOME->
AND NOT   M00723	// R_4th BD Z NOT MV
NOT
OUT       M0162C	// R_1-2 ROT R HOLD CUT
; L259
LOAD NOT  M03120	// R_4th Z IDLE POS ->
AND NOT   M03121	// R_4th Z CENTER POS ->
AND NOT   M03122	// R_4th Z BENDING POS ->
AND NOT   M03123	// R_4th Z BENDING POS 2 ->
AND NOT   M03124	// -
AND NOT   M03125	// -
AND NOT   M0312A	// -
AND NOT   M01625	// R_1-2 ROT R INITIAL ->
NOT
OUTP      M0162D	// R_1-2 ROT R START 1PLS
; L260
LOAD      D001380.7	// R_4th BD Z inposition
OUTP      M0162E	// R_1-2 ROT R POS OK PLS

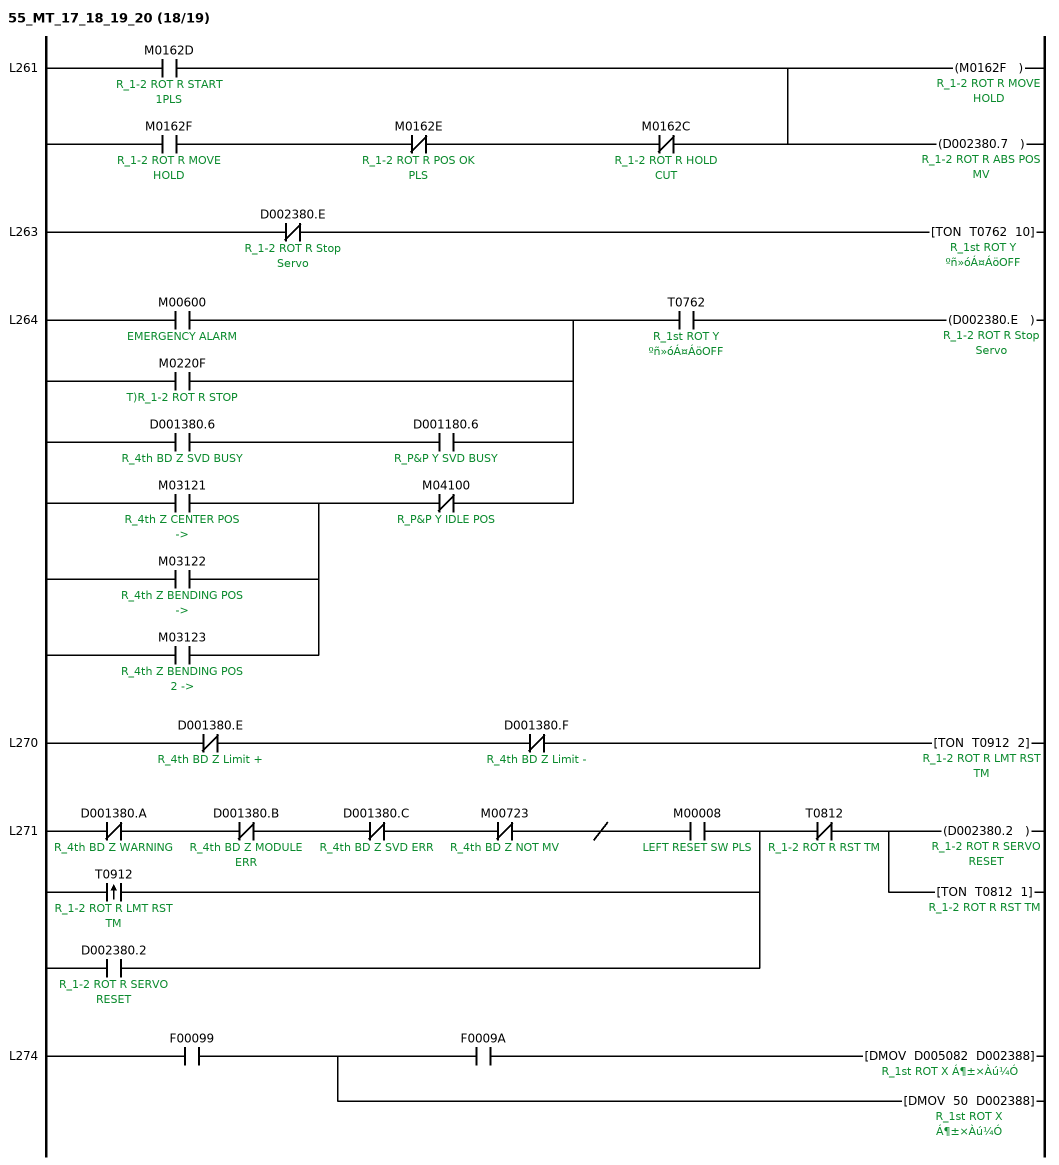
; L261
LOAD      M0162D	// R_1-2 ROT R START 1PLS
LOAD      M0162F	// R_1-2 ROT R MOVE HOLD
AND NOT   M0162E	// R_1-2 ROT R POS OK PLS
AND NOT   M0162C	// R_1-2 ROT R HOLD CUT
OR LOAD
OUT       M0162F	// R_1-2 ROT R MOVE HOLD
OUT       D002380.7	// R_1-2 ROT R ABS POS MV
; L263
LOAD NOT  D002380.E	// R_1-2 ROT R Stop Servo
TON       T0762 10	// R_1st ROT Y ºñ»óÁ¤ÁöOFF
; L264
LOAD      M00600	// EMERGENCY ALARM
OR        M0220F	// T)R_1-2 ROT R STOP
LOAD      D001380.6	// R_4th BD Z SVD BUSY
AND       D001180.6	// R_P&P Y SVD BUSY
OR LOAD
LOAD      M03121	// R_4th Z CENTER POS ->
OR        M03122	// R_4th Z BENDING POS ->
OR        M03123	// R_4th Z BENDING POS 2 ->
AND NOT   M04100	// R_P&P Y IDLE POS
OR LOAD
AND       T0762	// R_1st ROT Y ºñ»óÁ¤ÁöOFF
OUT       D002380.E	// R_1-2 ROT R Stop Servo
; L270
LOAD NOT  D001380.E	// R_4th BD Z Limit +
AND NOT   D001380.F	// R_4th BD Z Limit -
TON       T0912 2	// R_1-2 ROT R LMT RST TM
; L271
LOAD NOT  D001380.A	// R_4th BD Z WARNING
AND NOT   D001380.B	// R_4th BD Z MODULE ERR
AND NOT   D001380.C	// R_4th BD Z SVD ERR
AND NOT   M00723	// R_4th BD Z NOT MV
NOT
AND       M00008	// LEFT RESET SW PLS
ORP       T0912	// R_1-2 ROT R LMT RST TM
OR        D002380.2	// R_1-2 ROT R SERVO RESET
AND NOT   T0812	// R_1-2 ROT R RST TM
OUT       D002380.2	// R_1-2 ROT R SERVO RESET
TON       T0812 1	// R_1-2 ROT R RST TM
; L274
LOAD      F00099
MPUSH
AND       F0009A
DMOV      D005082 D002388	// R_1st ROT X Á¶±×Àú¼Ó
MPOP
DMOV      50 D002388	// R_1st ROT X Á¶±×Àú¼Ó

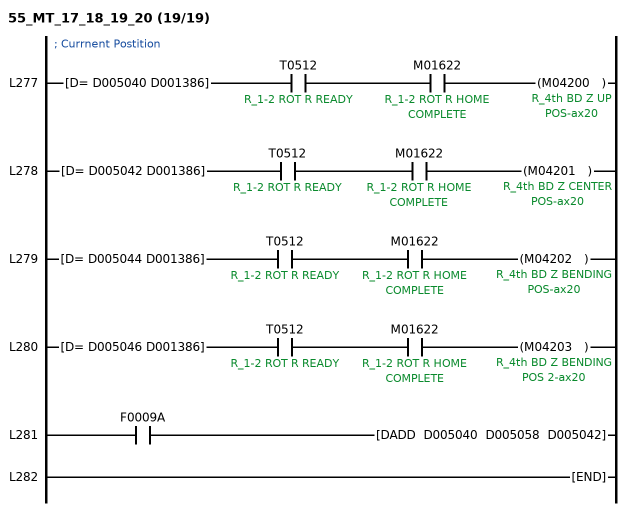
// Currnent Postition
; L277
LOADD=    D005040 D001386
AND       T0512	// R_1-2 ROT R READY
AND       M01622	// R_1-2 ROT R HOME COMPLETE
OUT       M04200	// R_4th BD Z UP POS-ax20
; L278
LOADD=    D005042 D001386
AND       T0512	// R_1-2 ROT R READY
AND       M01622	// R_1-2 ROT R HOME COMPLETE
OUT       M04201	// R_4th BD Z CENTER POS-ax20
; L279
LOADD=    D005044 D001386
AND       T0512	// R_1-2 ROT R READY
AND       M01622	// R_1-2 ROT R HOME COMPLETE
OUT       M04202	// R_4th BD Z BENDING POS-ax20
; L280
LOADD=    D005046 D001386
AND       T0512	// R_1-2 ROT R READY
AND       M01622	// R_1-2 ROT R HOME COMPLETE
OUT       M04203	// R_4th BD Z BENDING POS 2-ax20
; L281
LOAD      F0009A
DADD      D005040 D005058 D005042
; L282
END

PROGRAM 81_OUTPUT (task: ½ºÄµ ÇÁ·Î±×·¥)

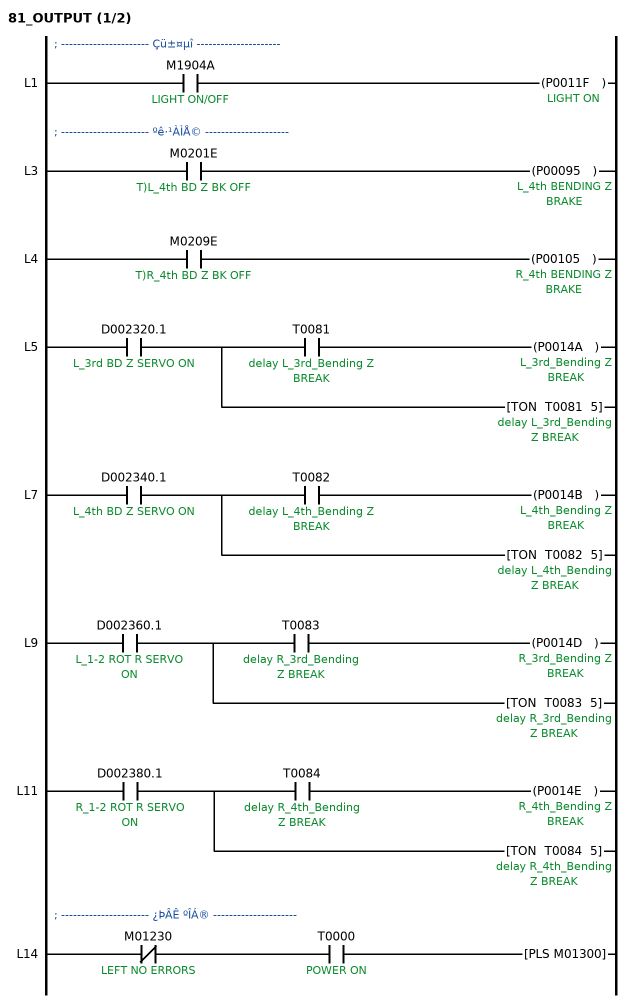
// ---------------------- Çü±¤µî ---------------------
; L1
LOAD      M1904A	// LIGHT ON/OFF
OUT       P0011F	// LIGHT ON
// ---------------------- ºê·¹ÀÌÅ© ---------------------
; L3
LOAD      M0201E	// T)L_4th BD Z BK OFF
OUT       P00095	// L_4th BENDING Z BRAKE
; L4
LOAD      M0209E	// T)R_4th BD Z BK OFF
OUT       P00105	// R_4th BENDING Z BRAKE
; L5
LOAD      D002320.1	// L_3rd BD Z SERVO ON
MPUSH
AND       T0081	// delay L_3rd_Bending Z BREAK
OUT       P0014A	// L_3rd_Bending Z BREAK
MPOP
TON       T0081 5	// delay L_3rd_Bending Z BREAK
; L7
LOAD      D002340.1	// L_4th BD Z SERVO ON
MPUSH
AND       T0082	// delay L_4th_Bending Z BREAK
OUT       P0014B	// L_4th_Bending Z BREAK
MPOP
TON       T0082 5	// delay L_4th_Bending Z BREAK
; L9
LOAD      D002360.1	// L_1-2 ROT R SERVO ON
MPUSH
AND       T0083	// delay R_3rd_Bending Z BREAK
OUT       P0014D	// R_3rd_Bending Z BREAK
MPOP
TON       T0083 5	// delay R_3rd_Bending Z BREAK
; L11
LOAD      D002380.1	// R_1-2 ROT R SERVO ON
MPUSH
AND       T0084	// delay R_4th_Bending Z BREAK
OUT       P0014E	// R_4th_Bending Z BREAK
MPOP
TON       T0084 5	// delay R_4th_Bending Z BREAK
// ---------------------- ¿ÞÂÊ ºÎÁ® ---------------------
; L14
LOAD NOT  M01230	// LEFT NO ERRORS
AND       T0000	// POWER ON
OUTP      M01300

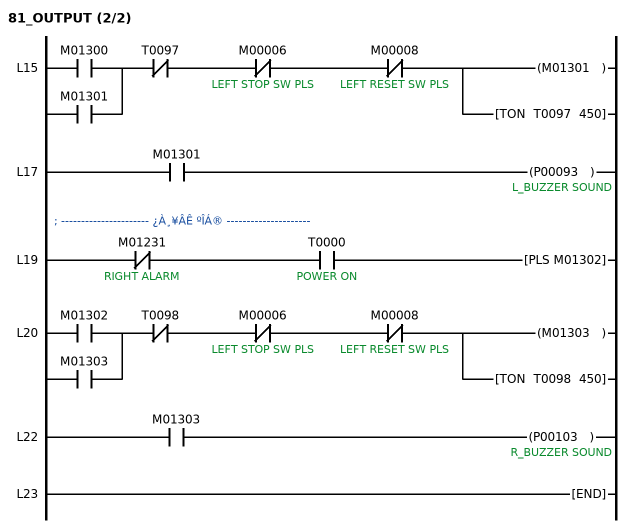
; L15
LOAD      M01300
OR        M01301
AND NOT   T0097
AND NOT   M00006	// LEFT STOP SW PLS
AND NOT   M00008	// LEFT RESET SW PLS
OUT       M01301
TON       T0097 450
; L17
LOAD      M01301
OUT       P00093	// L_BUZZER SOUND
// ---------------------- ¿À¸¥ÂÊ ºÎÁ® ---------------------
; L19
LOAD NOT  M01231	// RIGHT ALARM
AND       T0000	// POWER ON
OUTP      M01302
; L20
LOAD      M01302
OR        M01303
AND NOT   T0098
AND NOT   M00006	// LEFT STOP SW PLS
AND NOT   M00008	// LEFT RESET SW PLS
OUT       M01303
TON       T0098 450
; L22
LOAD      M01303
OUT       P00103	// R_BUZZER SOUND
; L23
END

PROGRAM 82_L_MANUAL (task: ½ºÄµ ÇÁ·Î±×·¥)

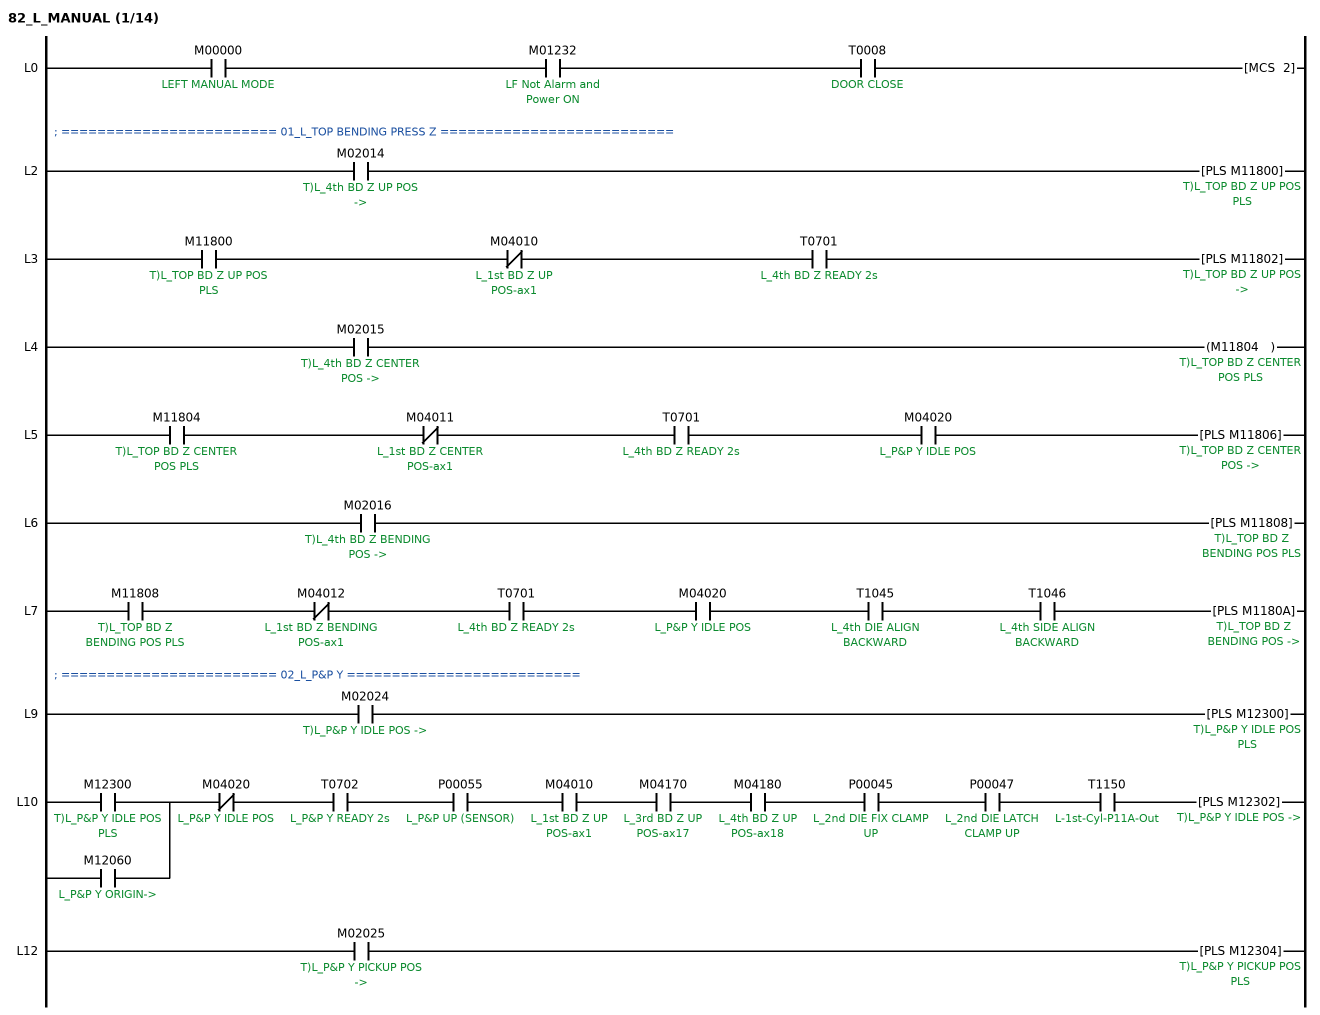
; L0
LOAD      M00000	// LEFT MANUAL MODE
AND       M01232	// LF Not Alarm and Power ON
AND       T0008	// DOOR CLOSE
MCS       2
// ======================== 01_L_TOP BENDING PRESS Z ==========================
; L2
LOAD      M02014	// T)L_4th BD Z UP POS ->
OUTP      M11800	// T)L_TOP BD Z UP POS PLS
; L3
LOAD      M11800	// T)L_TOP BD Z UP POS PLS
AND NOT   M04010	// L_1st BD Z UP POS-ax1
AND       T0701	// L_4th BD Z READY 2s
OUTP      M11802	// T)L_TOP BD Z UP POS ->
; L4
LOAD      M02015	// T)L_4th BD Z CENTER POS ->
OUT       M11804	// T)L_TOP BD Z CENTER POS PLS
; L5
LOAD      M11804	// T)L_TOP BD Z CENTER POS PLS
AND NOT   M04011	// L_1st BD Z CENTER POS-ax1
AND       T0701	// L_4th BD Z READY 2s
AND       M04020	// L_P&P Y IDLE POS
OUTP      M11806	// T)L_TOP BD Z CENTER POS ->
; L6
LOAD      M02016	// T)L_4th BD Z BENDING POS ->
OUTP      M11808	// T)L_TOP BD Z BENDING POS PLS
; L7
LOAD      M11808	// T)L_TOP BD Z BENDING POS PLS
AND NOT   M04012	// L_1st BD Z BENDING POS-ax1
AND       T0701	// L_4th BD Z READY 2s
AND       M04020	// L_P&P Y IDLE POS
AND       T1045	// L_4th DIE ALIGN BACKWARD
AND       T1046	// L_4th SIDE ALIGN BACKWARD
OUTP      M1180A	// T)L_TOP BD Z BENDING POS ->
// ======================== 02_L_P&P Y ==========================
; L9
LOAD      M02024	// T)L_P&P Y IDLE POS ->
OUTP      M12300	// T)L_P&P Y IDLE POS PLS
; L10
LOAD      M12300	// T)L_P&P Y IDLE POS PLS
OR        M12060	// L_P&P Y ORIGIN->
AND NOT   M04020	// L_P&P Y IDLE POS
AND       T0702	// L_P&P Y READY 2s
AND       P00055	// L_P&P UP (SENSOR)
AND       M04010	// L_1st BD Z UP POS-ax1
AND       M04170	// L_3rd BD Z UP POS-ax17
AND       M04180	// L_4th BD Z UP POS-ax18
AND       P00045	// L_2nd DIE FIX CLAMP UP
AND       P00047	// L_2nd DIE LATCH CLAMP UP
AND       T1150	// L-1st-Cyl-P11A-Out
OUTP      M12302	// T)L_P&P Y IDLE POS ->
; L12
LOAD      M02025	// T)L_P&P Y PICKUP POS ->
OUTP      M12304	// T)L_P&P Y PICKUP POS PLS

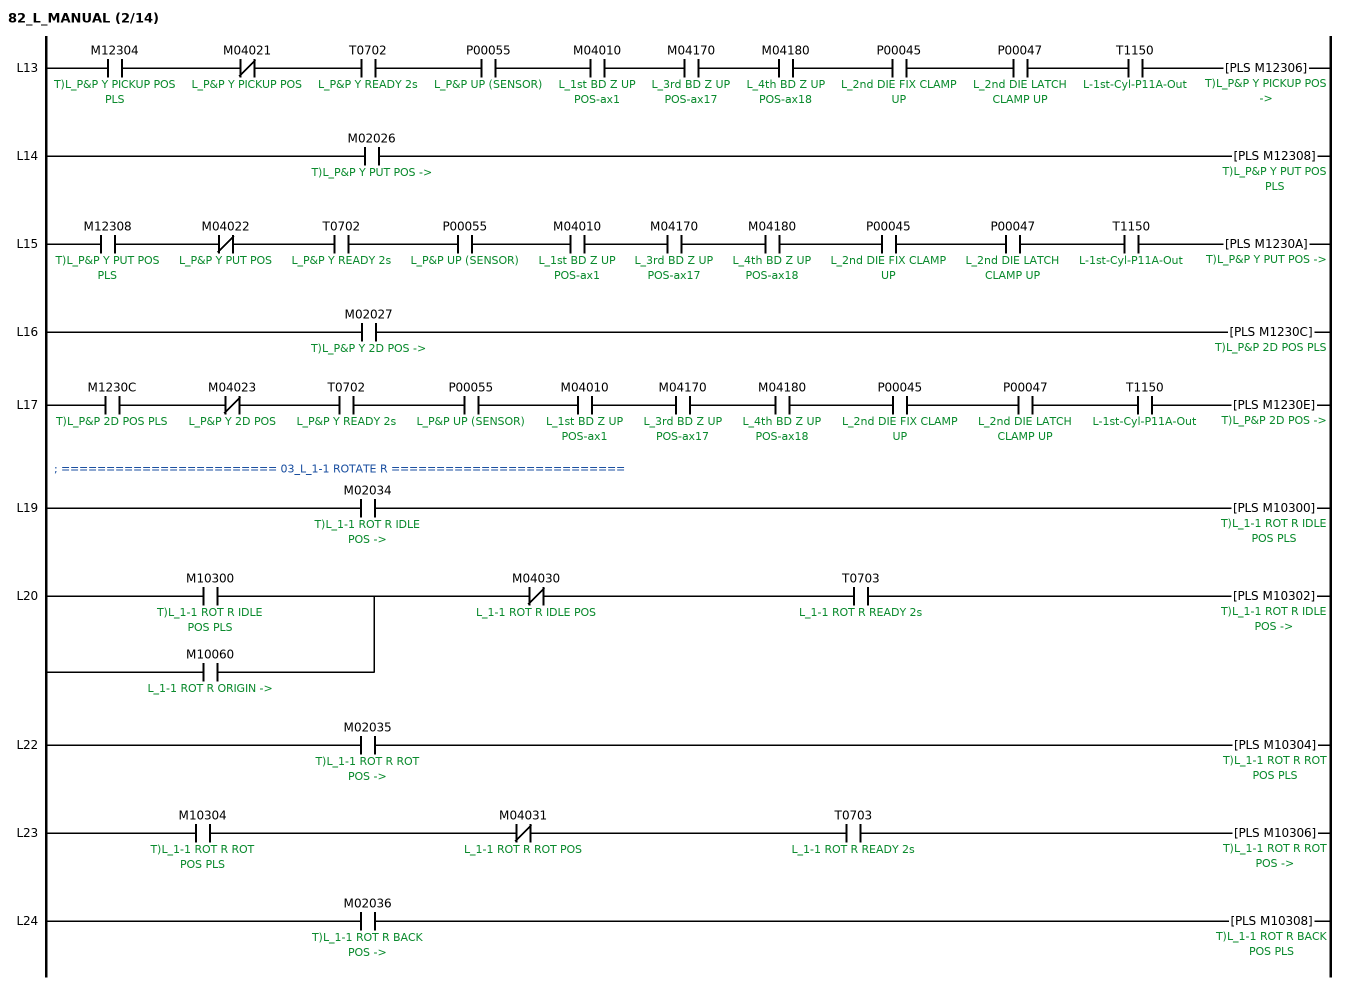
; L13
LOAD      M12304	// T)L_P&P Y PICKUP POS PLS
AND NOT   M04021	// L_P&P Y PICKUP POS
AND       T0702	// L_P&P Y READY 2s
AND       P00055	// L_P&P UP (SENSOR)
AND       M04010	// L_1st BD Z UP POS-ax1
AND       M04170	// L_3rd BD Z UP POS-ax17
AND       M04180	// L_4th BD Z UP POS-ax18
AND       P00045	// L_2nd DIE FIX CLAMP UP
AND       P00047	// L_2nd DIE LATCH CLAMP UP
AND       T1150	// L-1st-Cyl-P11A-Out
OUTP      M12306	// T)L_P&P Y PICKUP POS ->
; L14
LOAD      M02026	// T)L_P&P Y PUT POS ->
OUTP      M12308	// T)L_P&P Y PUT POS PLS
; L15
LOAD      M12308	// T)L_P&P Y PUT POS PLS
AND NOT   M04022	// L_P&P Y PUT POS
AND       T0702	// L_P&P Y READY 2s
AND       P00055	// L_P&P UP (SENSOR)
AND       M04010	// L_1st BD Z UP POS-ax1
AND       M04170	// L_3rd BD Z UP POS-ax17
AND       M04180	// L_4th BD Z UP POS-ax18
AND       P00045	// L_2nd DIE FIX CLAMP UP
AND       P00047	// L_2nd DIE LATCH CLAMP UP
AND       T1150	// L-1st-Cyl-P11A-Out
OUTP      M1230A	// T)L_P&P Y PUT POS ->
; L16
LOAD      M02027	// T)L_P&P Y 2D POS ->
OUTP      M1230C	// T)L_P&P 2D POS PLS
; L17
LOAD      M1230C	// T)L_P&P 2D POS PLS
AND NOT   M04023	// L_P&P Y 2D POS
AND       T0702	// L_P&P Y READY 2s
AND       P00055	// L_P&P UP (SENSOR)
AND       M04010	// L_1st BD Z UP POS-ax1
AND       M04170	// L_3rd BD Z UP POS-ax17
AND       M04180	// L_4th BD Z UP POS-ax18
AND       P00045	// L_2nd DIE FIX CLAMP UP
AND       P00047	// L_2nd DIE LATCH CLAMP UP
AND       T1150	// L-1st-Cyl-P11A-Out
OUTP      M1230E	// T)L_P&P 2D POS ->
// ======================== 03_L_1-1 ROTATE R ==========================
; L19
LOAD      M02034	// T)L_1-1 ROT R IDLE POS ->
OUTP      M10300	// T)L_1-1 ROT R IDLE POS PLS
; L20
LOAD      M10300	// T)L_1-1 ROT R IDLE POS PLS
OR        M10060	// L_1-1 ROT R ORIGIN ->
AND NOT   M04030	// L_1-1 ROT R IDLE POS
AND       T0703	// L_1-1 ROT R READY 2s
OUTP      M10302	// T)L_1-1 ROT R IDLE POS ->
; L22
LOAD      M02035	// T)L_1-1 ROT R ROT POS ->
OUTP      M10304	// T)L_1-1 ROT R ROT POS PLS
; L23
LOAD      M10304	// T)L_1-1 ROT R ROT POS PLS
AND NOT   M04031	// L_1-1 ROT R ROT POS
AND       T0703	// L_1-1 ROT R READY 2s
OUTP      M10306	// T)L_1-1 ROT R ROT POS ->
; L24
LOAD      M02036	// T)L_1-1 ROT R BACK POS ->
OUTP      M10308	// T)L_1-1 ROT R BACK POS PLS

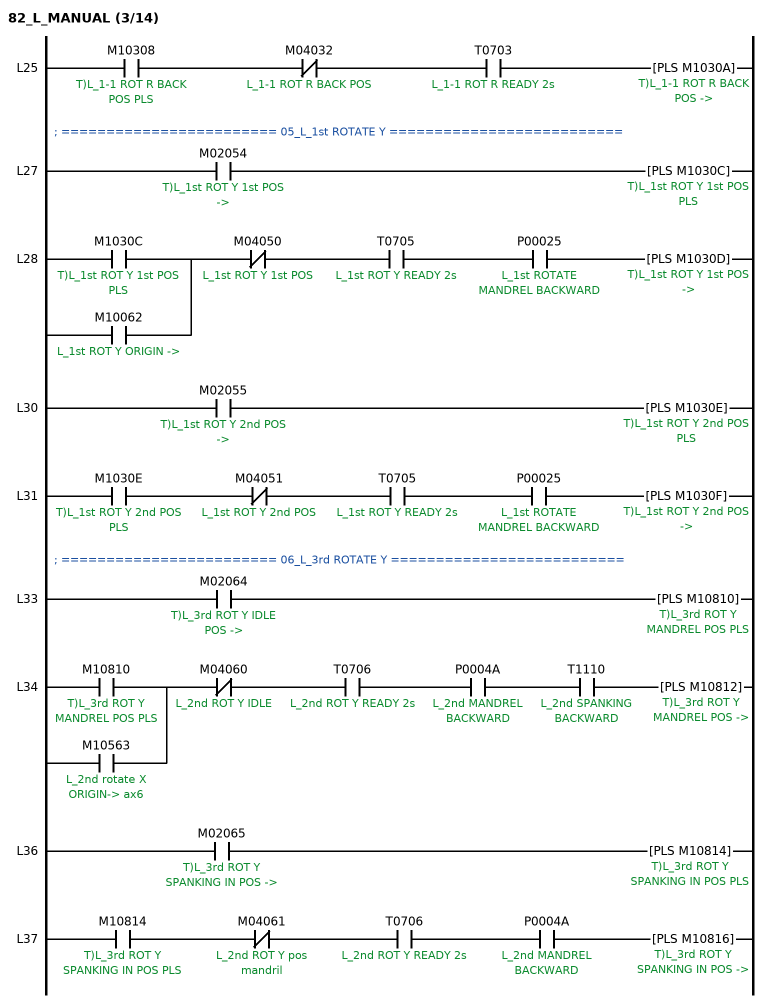
; L25
LOAD      M10308	// T)L_1-1 ROT R BACK POS PLS
AND NOT   M04032	// L_1-1 ROT R BACK POS
AND       T0703	// L_1-1 ROT R READY 2s
OUTP      M1030A	// T)L_1-1 ROT R BACK POS ->
// ======================== 05_L_1st ROTATE Y ==========================
; L27
LOAD      M02054	// T)L_1st ROT Y 1st POS ->
OUTP      M1030C	// T)L_1st ROT Y 1st POS PLS
; L28
LOAD      M1030C	// T)L_1st ROT Y 1st POS PLS
OR        M10062	// L_1st ROT Y ORIGIN ->
AND NOT   M04050	// L_1st ROT Y 1st POS
AND       T0705	// L_1st ROT Y READY 2s
AND       P00025	// L_1st ROTATE MANDREL BACKWARD
OUTP      M1030D	// T)L_1st ROT Y 1st POS ->
; L30
LOAD      M02055	// T)L_1st ROT Y 2nd POS ->
OUTP      M1030E	// T)L_1st ROT Y 2nd POS PLS
; L31
LOAD      M1030E	// T)L_1st ROT Y 2nd POS PLS
AND NOT   M04051	// L_1st ROT Y 2nd POS
AND       T0705	// L_1st ROT Y READY 2s
AND       P00025	// L_1st ROTATE MANDREL BACKWARD
OUTP      M1030F	// T)L_1st ROT Y 2nd POS ->
// ======================== 06_L_3rd ROTATE Y ==========================
; L33
LOAD      M02064	// T)L_3rd ROT Y IDLE POS ->
OUTP      M10810	// T)L_3rd ROT Y MANDREL POS PLS
; L34
LOAD      M10810	// T)L_3rd ROT Y MANDREL POS PLS
OR        M10563	// L_2nd rotate X ORIGIN-> ax6
AND NOT   M04060	// L_2nd ROT Y IDLE
AND       T0706	// L_2nd ROT Y READY 2s
AND       P0004A	// L_2nd MANDREL BACKWARD
AND       T1110	// L_2nd SPANKING BACKWARD
OUTP      M10812	// T)L_3rd ROT Y MANDREL POS ->
; L36
LOAD      M02065	// T)L_3rd ROT Y SPANKING IN POS ->
OUTP      M10814	// T)L_3rd ROT Y SPANKING IN POS PLS
; L37
LOAD      M10814	// T)L_3rd ROT Y SPANKING IN POS PLS
AND NOT   M04061	// L_2nd ROT Y pos mandril
AND       T0706	// L_2nd ROT Y READY 2s
AND       P0004A	// L_2nd MANDREL BACKWARD
OUTP      M10816	// T)L_3rd ROT Y SPANKING IN POS ->

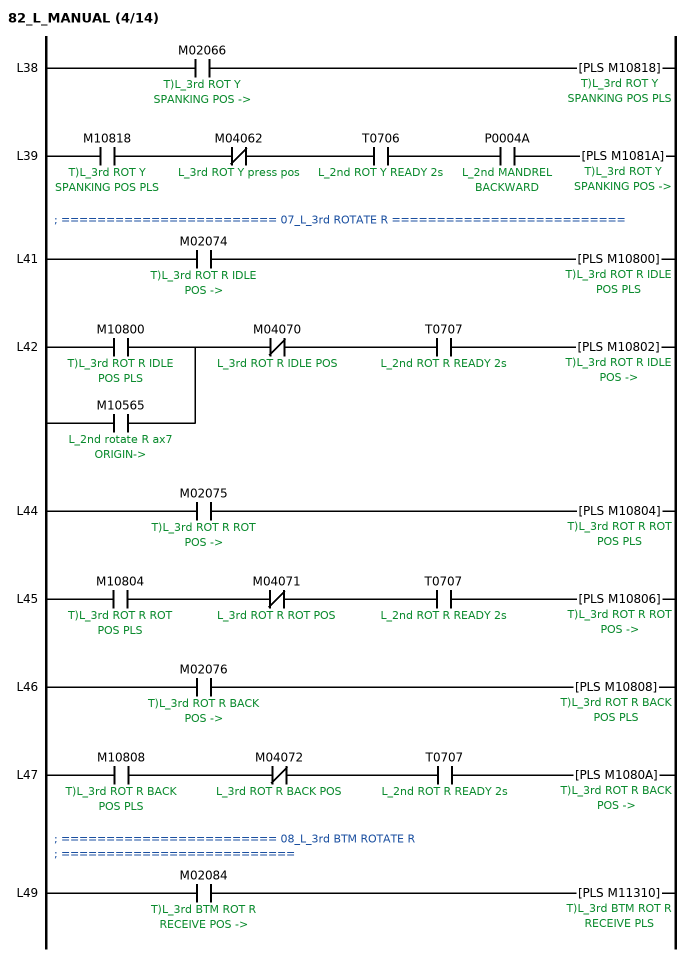
; L38
LOAD      M02066	// T)L_3rd ROT Y SPANKING POS ->
OUTP      M10818	// T)L_3rd ROT Y SPANKING POS PLS
; L39
LOAD      M10818	// T)L_3rd ROT Y SPANKING POS PLS
AND NOT   M04062	// L_3rd ROT Y press pos
AND       T0706	// L_2nd ROT Y READY 2s
AND       P0004A	// L_2nd MANDREL BACKWARD
OUTP      M1081A	// T)L_3rd ROT Y SPANKING POS ->
// ======================== 07_L_3rd ROTATE R ==========================
; L41
LOAD      M02074	// T)L_3rd ROT R IDLE POS ->
OUTP      M10800	// T)L_3rd ROT R IDLE POS PLS
; L42
LOAD      M10800	// T)L_3rd ROT R IDLE POS PLS
OR        M10565	// L_2nd rotate R ax7 ORIGIN->
AND NOT   M04070	// L_3rd ROT R IDLE POS
AND       T0707	// L_2nd ROT R READY 2s
OUTP      M10802	// T)L_3rd ROT R IDLE POS ->
; L44
LOAD      M02075	// T)L_3rd ROT R ROT POS ->
OUTP      M10804	// T)L_3rd ROT R ROT POS PLS
; L45
LOAD      M10804	// T)L_3rd ROT R ROT POS PLS
AND NOT   M04071	// L_3rd ROT R ROT POS
AND       T0707	// L_2nd ROT R READY 2s
OUTP      M10806	// T)L_3rd ROT R ROT POS ->
; L46
LOAD      M02076	// T)L_3rd ROT R BACK POS ->
OUTP      M10808	// T)L_3rd ROT R BACK POS PLS
; L47
LOAD      M10808	// T)L_3rd ROT R BACK POS PLS
AND NOT   M04072	// L_3rd ROT R BACK POS
AND       T0707	// L_2nd ROT R READY 2s
OUTP      M1080A	// T)L_3rd ROT R BACK POS ->
// ======================== 08_L_3rd BTM ROTATE R ==========================
; L49
LOAD      M02084	// T)L_3rd BTM ROT R RECEIVE POS ->
OUTP      M11310	// T)L_3rd BTM ROT R RECEIVE PLS

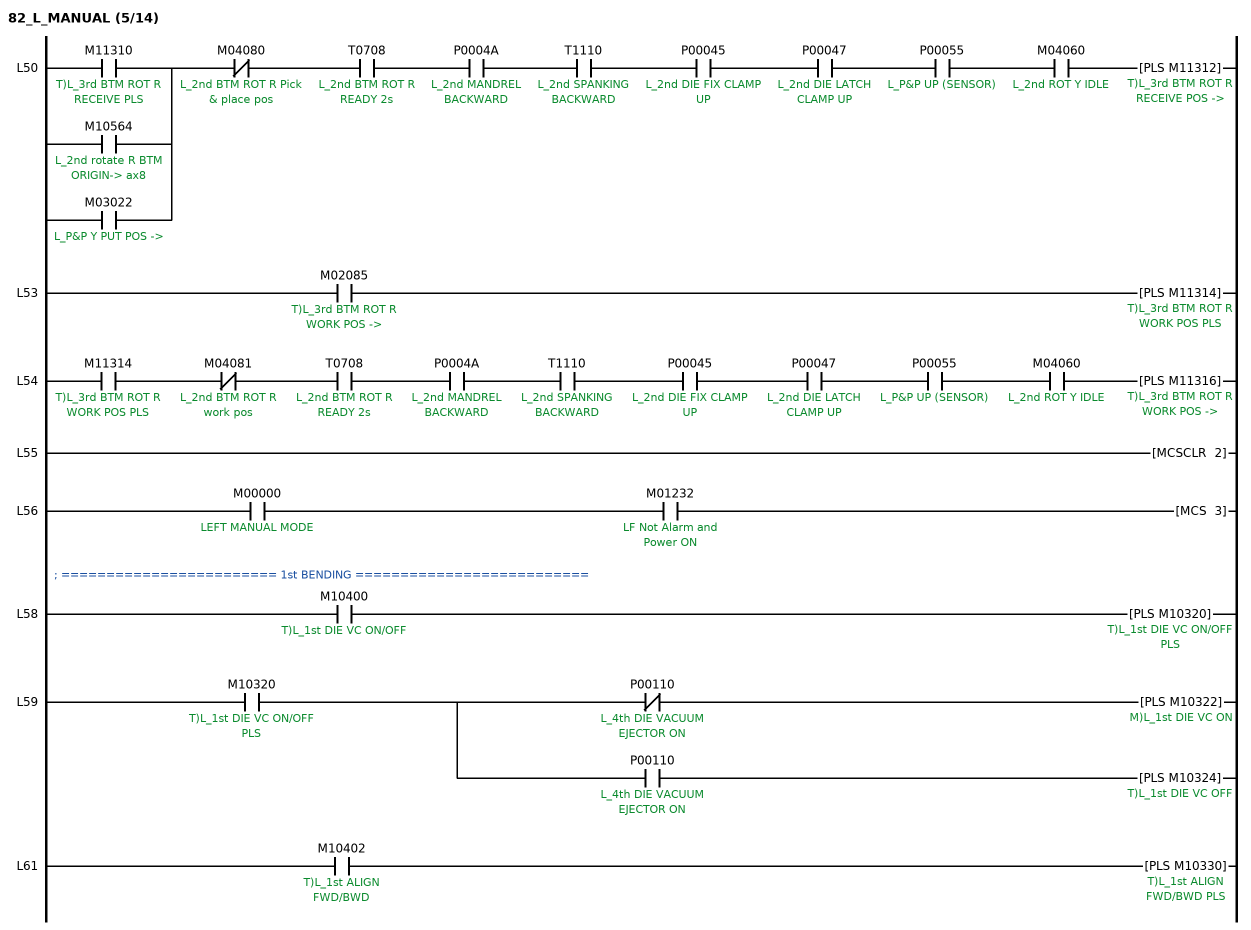
; L50
LOAD      M11310	// T)L_3rd BTM ROT R RECEIVE PLS
OR        M10564	// L_2nd rotate R BTM  ORIGIN-> ax8
OR        M03022	// L_P&P Y PUT POS ->
AND NOT   M04080	// L_2nd BTM ROT R Pick & place pos
AND       T0708	// L_2nd BTM ROT R READY 2s
AND       P0004A	// L_2nd MANDREL BACKWARD
AND       T1110	// L_2nd SPANKING BACKWARD
AND       P00045	// L_2nd DIE FIX CLAMP UP
AND       P00047	// L_2nd DIE LATCH CLAMP UP
AND       P00055	// L_P&P UP (SENSOR)
AND       M04060	// L_2nd ROT Y IDLE
OUTP      M11312	// T)L_3rd BTM ROT R RECEIVE POS ->
; L53
LOAD      M02085	// T)L_3rd BTM ROT R WORK POS ->
OUTP      M11314	// T)L_3rd BTM ROT R WORK POS PLS
; L54
LOAD      M11314	// T)L_3rd BTM ROT R WORK POS PLS
AND NOT   M04081	// L_2nd BTM ROT R work pos
AND       T0708	// L_2nd BTM ROT R READY 2s
AND       P0004A	// L_2nd MANDREL BACKWARD
AND       T1110	// L_2nd SPANKING BACKWARD
AND       P00045	// L_2nd DIE FIX CLAMP UP
AND       P00047	// L_2nd DIE LATCH CLAMP UP
AND       P00055	// L_P&P UP (SENSOR)
AND       M04060	// L_2nd ROT Y IDLE
OUTP      M11316	// T)L_3rd BTM ROT R WORK POS ->
; L55
MCSCLR    2
; L56
LOAD      M00000	// LEFT MANUAL MODE
AND       M01232	// LF Not Alarm and Power ON
MCS       3
// ======================== 1st BENDING ==========================
; L58
LOAD      M10400	// T)L_1st DIE VC ON/OFF
OUTP      M10320	// T)L_1st DIE VC ON/OFF PLS
; L59
LOAD      M10320	// T)L_1st DIE VC ON/OFF PLS
MPUSH
AND NOT   P00110	// L_4th DIE VACUUM EJECTOR ON
OUTP      M10322	// M)L_1st DIE VC ON
MPOP
AND       P00110	// L_4th DIE VACUUM EJECTOR ON
OUTP      M10324	// T)L_1st DIE VC OFF
; L61
LOAD      M10402	// T)L_1st ALIGN FWD/BWD
OUTP      M10330	// T)L_1st ALIGN FWD/BWD PLS

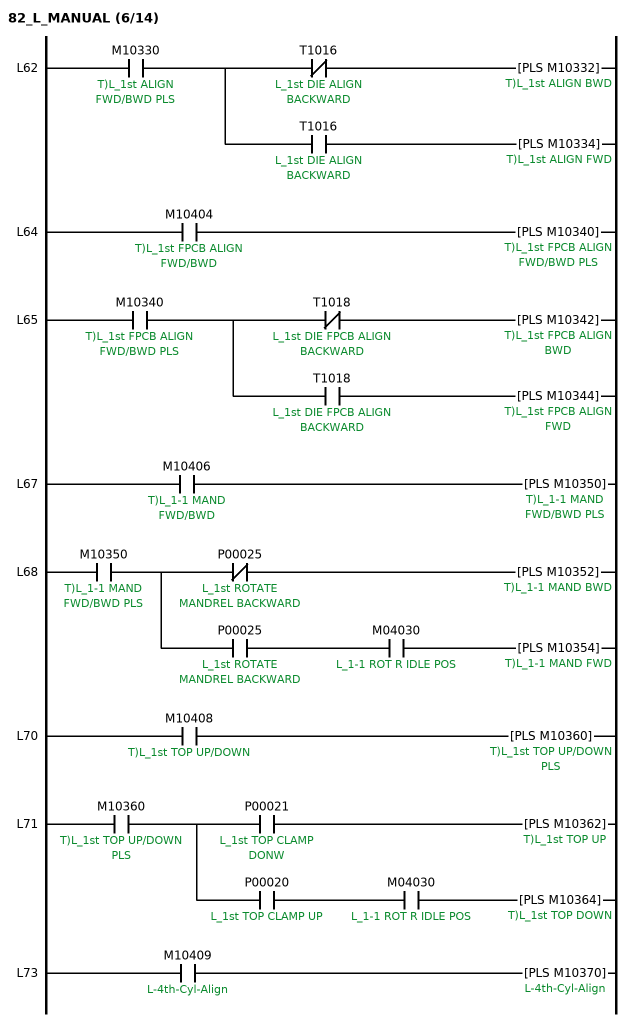
; L62
LOAD      M10330	// T)L_1st ALIGN FWD/BWD PLS
MPUSH
AND NOT   T1016	// L_1st DIE ALIGN BACKWARD
OUTP      M10332	// T)L_1st ALIGN BWD
MPOP
AND       T1016	// L_1st DIE ALIGN BACKWARD
OUTP      M10334	// T)L_1st ALIGN FWD
; L64
LOAD      M10404	// T)L_1st FPCB ALIGN FWD/BWD
OUTP      M10340	// T)L_1st FPCB ALIGN FWD/BWD PLS
; L65
LOAD      M10340	// T)L_1st FPCB ALIGN FWD/BWD PLS
MPUSH
AND NOT   T1018	// L_1st DIE FPCB ALIGN BACKWARD
OUTP      M10342	// T)L_1st FPCB ALIGN BWD
MPOP
AND       T1018	// L_1st DIE FPCB ALIGN BACKWARD
OUTP      M10344	// T)L_1st FPCB ALIGN FWD
; L67
LOAD      M10406	// T)L_1-1 MAND FWD/BWD
OUTP      M10350	// T)L_1-1 MAND FWD/BWD PLS
; L68
LOAD      M10350	// T)L_1-1 MAND FWD/BWD PLS
MPUSH
AND NOT   P00025	// L_1st ROTATE MANDREL BACKWARD
OUTP      M10352	// T)L_1-1 MAND BWD
MPOP
AND       P00025	// L_1st ROTATE MANDREL BACKWARD
AND       M04030	// L_1-1 ROT R IDLE POS
OUTP      M10354	// T)L_1-1 MAND FWD
; L70
LOAD      M10408	// T)L_1st TOP UP/DOWN
OUTP      M10360	// T)L_1st TOP UP/DOWN PLS
; L71
LOAD      M10360	// T)L_1st TOP UP/DOWN PLS
MPUSH
AND       P00021	// L_1st TOP CLAMP DONW
OUTP      M10362	// T)L_1st TOP UP
MPOP
AND       P00020	// L_1st TOP CLAMP UP
AND       M04030	// L_1-1 ROT R IDLE POS
OUTP      M10364	// T)L_1st TOP DOWN
; L73
LOAD      M10409	// L-4th-Cyl-Align
OUTP      M10370	// L-4th-Cyl-Align

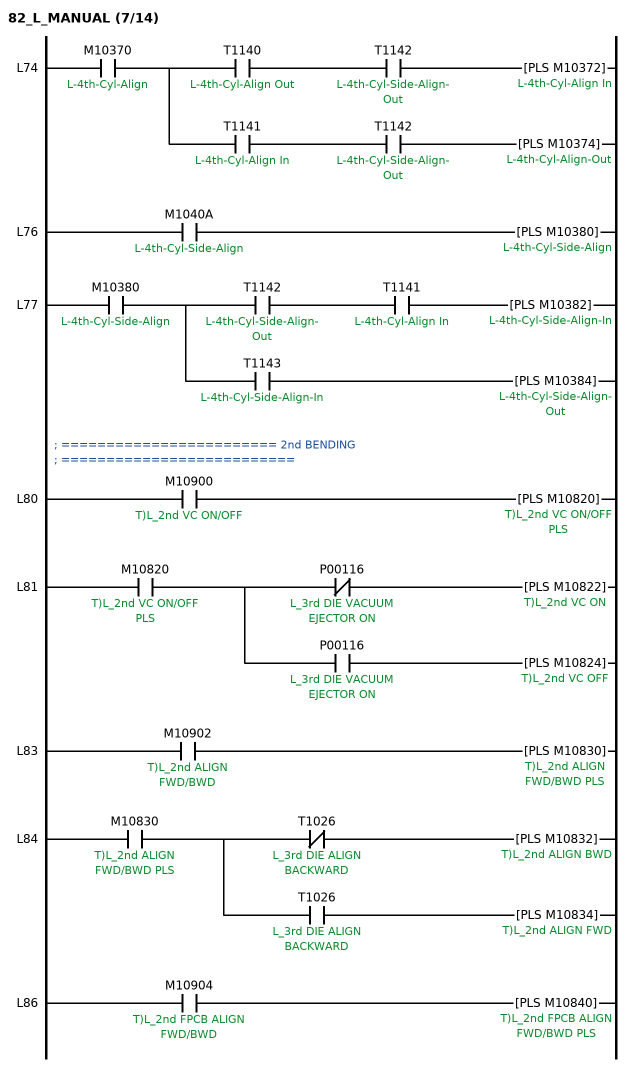
; L74
LOAD      M10370	// L-4th-Cyl-Align
MPUSH
AND       T1140	// L-4th-Cyl-Align Out
AND       T1142	// L-4th-Cyl-Side-Align-Out
OUTP      M10372	// L-4th-Cyl-Align In
MPOP
AND       T1141	// L-4th-Cyl-Align In
AND       T1142	// L-4th-Cyl-Side-Align-Out
OUTP      M10374	// L-4th-Cyl-Align-Out
; L76
LOAD      M1040A	// L-4th-Cyl-Side-Align
OUTP      M10380	// L-4th-Cyl-Side-Align
; L77
LOAD      M10380	// L-4th-Cyl-Side-Align
MPUSH
AND       T1142	// L-4th-Cyl-Side-Align-Out
AND       T1141	// L-4th-Cyl-Align In
OUTP      M10382	// L-4th-Cyl-Side-Align-In
MPOP
AND       T1143	// L-4th-Cyl-Side-Align-In
OUTP      M10384	// L-4th-Cyl-Side-Align-Out
// ======================== 2nd BENDING ==========================
; L80
LOAD      M10900	// T)L_2nd VC ON/OFF
OUTP      M10820	// T)L_2nd VC ON/OFF PLS
; L81
LOAD      M10820	// T)L_2nd VC ON/OFF PLS
MPUSH
AND NOT   P00116	// L_3rd DIE VACUUM EJECTOR ON
OUTP      M10822	// T)L_2nd VC ON
MPOP
AND       P00116	// L_3rd DIE VACUUM EJECTOR ON
OUTP      M10824	// T)L_2nd VC OFF
; L83
LOAD      M10902	// T)L_2nd ALIGN FWD/BWD
OUTP      M10830	// T)L_2nd ALIGN FWD/BWD PLS
; L84
LOAD      M10830	// T)L_2nd ALIGN FWD/BWD PLS
MPUSH
AND NOT   T1026	// L_3rd DIE ALIGN BACKWARD
OUTP      M10832	// T)L_2nd ALIGN BWD
MPOP
AND       T1026	// L_3rd DIE ALIGN BACKWARD
OUTP      M10834	// T)L_2nd ALIGN FWD
; L86
LOAD      M10904	// T)L_2nd FPCB ALIGN FWD/BWD
OUTP      M10840	// T)L_2nd FPCB ALIGN FWD/BWD PLS

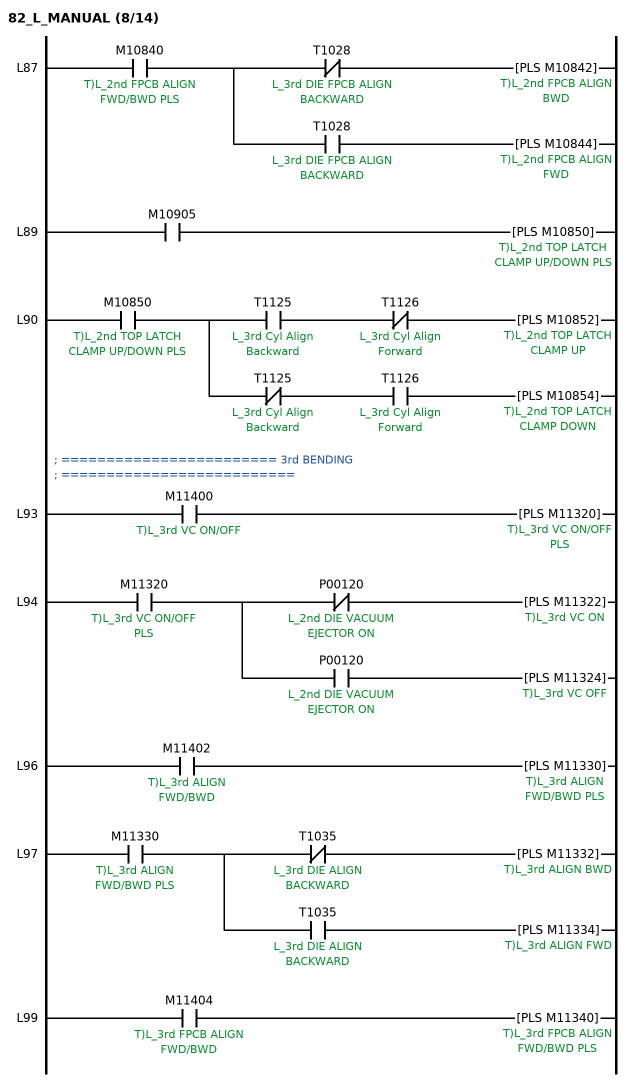
; L87
LOAD      M10840	// T)L_2nd FPCB ALIGN FWD/BWD PLS
MPUSH
AND NOT   T1028	// L_3rd DIE FPCB ALIGN BACKWARD
OUTP      M10842	// T)L_2nd FPCB ALIGN BWD
MPOP
AND       T1028	// L_3rd DIE FPCB ALIGN BACKWARD
OUTP      M10844	// T)L_2nd FPCB ALIGN FWD
; L89
LOAD      M10905
OUTP      M10850	// T)L_2nd TOP LATCH CLAMP UP/DOWN PLS
; L90
LOAD      M10850	// T)L_2nd TOP LATCH CLAMP UP/DOWN PLS
MPUSH
AND       T1125	// L_3rd Cyl Align Backward
AND NOT   T1126	// L_3rd Cyl Align Forward
OUTP      M10852	// T)L_2nd TOP LATCH CLAMP UP
MPOP
AND NOT   T1125	// L_3rd Cyl Align Backward
AND       T1126	// L_3rd Cyl Align Forward
OUTP      M10854	// T)L_2nd TOP LATCH CLAMP DOWN
// ======================== 3rd BENDING ==========================
; L93
LOAD      M11400	// T)L_3rd VC ON/OFF
OUTP      M11320	// T)L_3rd VC ON/OFF PLS
; L94
LOAD      M11320	// T)L_3rd VC ON/OFF PLS
MPUSH
AND NOT   P00120	// L_2nd DIE VACUUM EJECTOR ON
OUTP      M11322	// T)L_3rd VC ON
MPOP
AND       P00120	// L_2nd DIE VACUUM EJECTOR ON
OUTP      M11324	// T)L_3rd VC OFF
; L96
LOAD      M11402	// T)L_3rd ALIGN FWD/BWD
OUTP      M11330	// T)L_3rd ALIGN FWD/BWD PLS
; L97
LOAD      M11330	// T)L_3rd ALIGN FWD/BWD PLS
MPUSH
AND NOT   T1035	// L_3rd DIE ALIGN BACKWARD
OUTP      M11332	// T)L_3rd ALIGN BWD
MPOP
AND       T1035	// L_3rd DIE ALIGN BACKWARD
OUTP      M11334	// T)L_3rd ALIGN FWD
; L99
LOAD      M11404	// T)L_3rd FPCB ALIGN FWD/BWD
OUTP      M11340	// T)L_3rd FPCB ALIGN FWD/BWD PLS

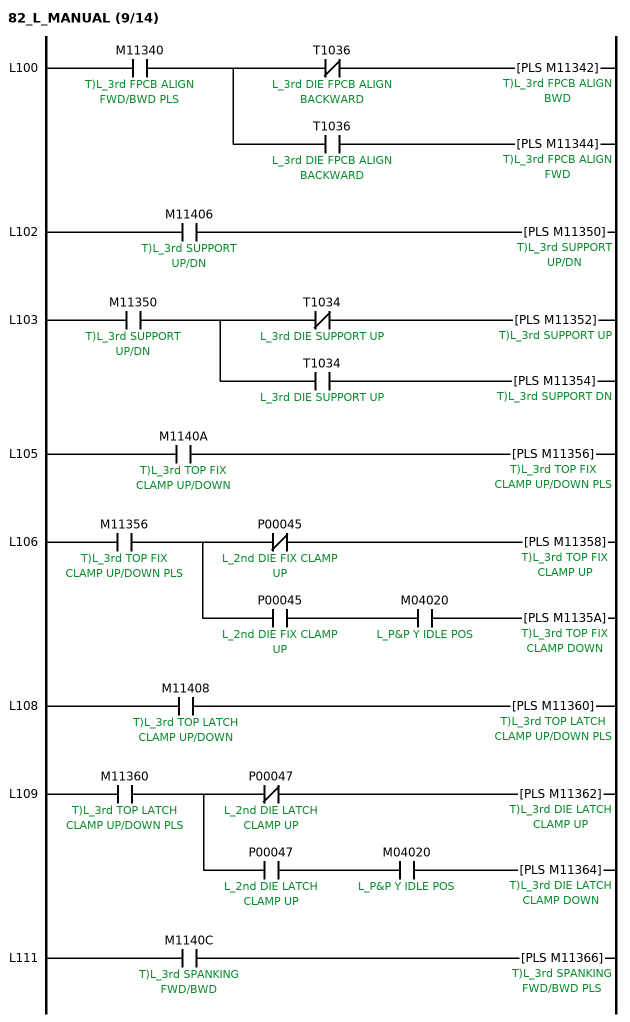
; L100
LOAD      M11340	// T)L_3rd FPCB ALIGN FWD/BWD PLS
MPUSH
AND NOT   T1036	// L_3rd DIE FPCB ALIGN BACKWARD
OUTP      M11342	// T)L_3rd FPCB ALIGN BWD
MPOP
AND       T1036	// L_3rd DIE FPCB ALIGN BACKWARD
OUTP      M11344	// T)L_3rd FPCB ALIGN FWD
; L102
LOAD      M11406	// T)L_3rd SUPPORT UP/DN
OUTP      M11350	// T)L_3rd SUPPORT UP/DN
; L103
LOAD      M11350	// T)L_3rd SUPPORT UP/DN
MPUSH
AND NOT   T1034	// L_3rd DIE SUPPORT UP
OUTP      M11352	// T)L_3rd SUPPORT UP
MPOP
AND       T1034	// L_3rd DIE SUPPORT UP
OUTP      M11354	// T)L_3rd SUPPORT DN
; L105
LOAD      M1140A	// T)L_3rd TOP FIX CLAMP UP/DOWN
OUTP      M11356	// T)L_3rd TOP FIX CLAMP UP/DOWN PLS
; L106
LOAD      M11356	// T)L_3rd TOP FIX CLAMP UP/DOWN PLS
MPUSH
AND NOT   P00045	// L_2nd DIE FIX CLAMP UP
OUTP      M11358	// T)L_3rd TOP FIX CLAMP UP
MPOP
AND       P00045	// L_2nd DIE FIX CLAMP UP
AND       M04020	// L_P&P Y IDLE POS
OUTP      M1135A	// T)L_3rd TOP FIX CLAMP DOWN
; L108
LOAD      M11408	// T)L_3rd TOP LATCH CLAMP UP/DOWN
OUTP      M11360	// T)L_3rd TOP LATCH CLAMP UP/DOWN PLS
; L109
LOAD      M11360	// T)L_3rd TOP LATCH CLAMP UP/DOWN PLS
MPUSH
AND NOT   P00047	// L_2nd DIE LATCH CLAMP UP
OUTP      M11362	// T)L_3rd DIE LATCH CLAMP UP
MPOP
AND       P00047	// L_2nd DIE LATCH CLAMP UP
AND       M04020	// L_P&P Y IDLE POS
OUTP      M11364	// T)L_3rd DIE LATCH CLAMP DOWN
; L111
LOAD      M1140C	// T)L_3rd SPANKING FWD/BWD
OUTP      M11366	// T)L_3rd SPANKING FWD/BWD PLS

